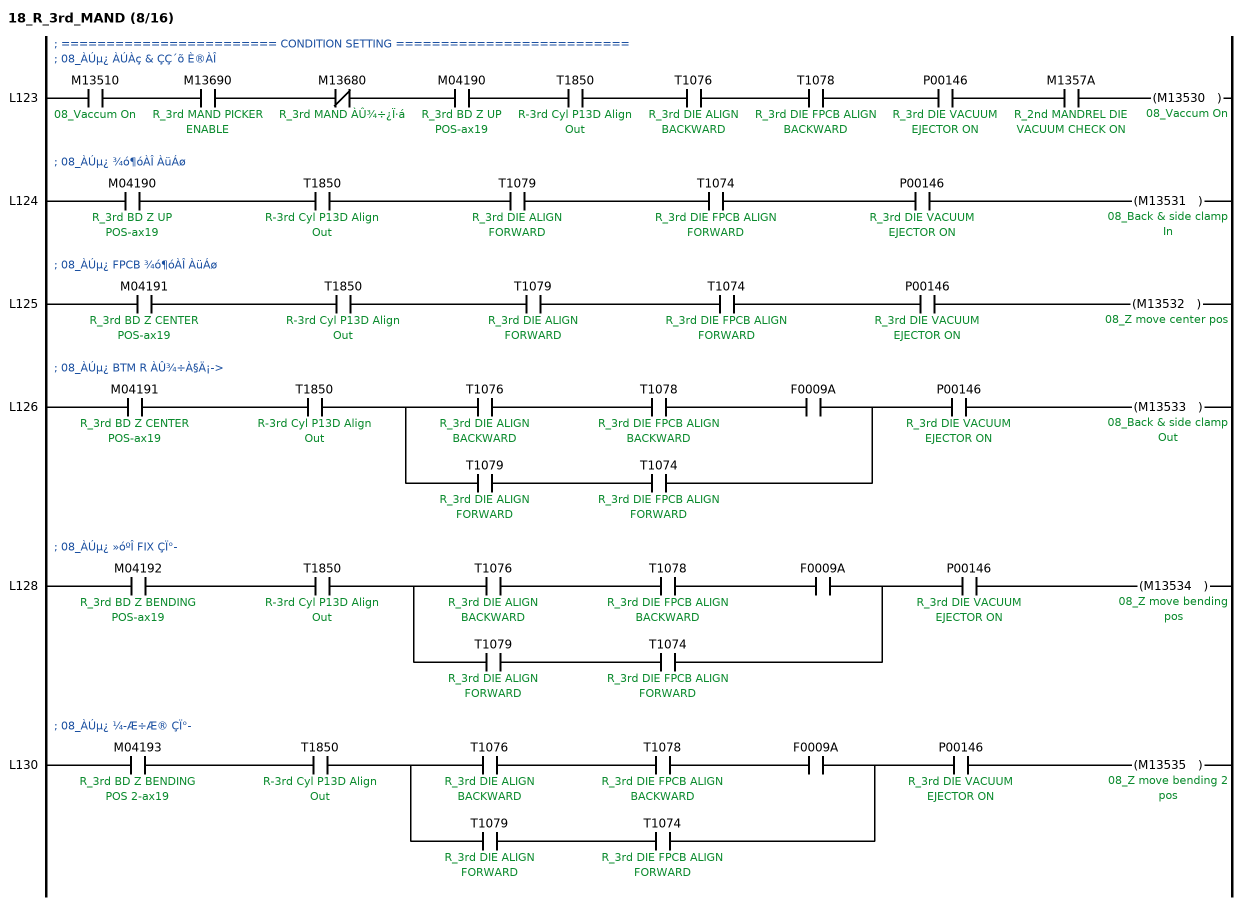
[picture p168: 18_R_3rd_MAND rungs L123-L130]
// ======================== CONDITION SETTING ==========================
; L123
LOAD      M13510	// 08_Vaccum On
AND       M13690	// R_3rd MAND PICKER ENABLE
AND NOT   M13680	// R_3rd MAND ÀÛ¾÷¿Ï·á
AND       M04190	// R_3rd BD Z UP POS-ax19
AND       T1850	// R-3rd Cyl P13D Align Out
AND       T1076	// R_3rd DIE ALIGN BACKWARD
AND       T1078	// R_3rd DIE FPCB ALIGN BACKWARD
AND       P00146	// R_3rd DIE VACUUM EJECTOR ON
AND       M1357A	// R_2nd MANDREL DIE VACUUM CHECK ON
OUT       M13530	// 08_Vaccum On
// output comment: 08_ÀÚµ¿ ÀÚÀç & ÇÇ´õ È®ÀÎ
; L124
LOAD      M04190	// R_3rd BD Z UP POS-ax19
AND       T1850	// R-3rd Cyl P13D Align Out
AND       T1079	// R_3rd DIE ALIGN FORWARD
AND       T1074	// R_3rd DIE FPCB ALIGN FORWARD
AND       P00146	// R_3rd DIE VACUUM EJECTOR ON
OUT       M13531	// 08_Back & side clamp In
// output comment: 08_ÀÚµ¿ ¾ó¶óÀÎ ÀüÁø
; L125
LOAD      M04191	// R_3rd BD Z CENTER POS-ax19
AND       T1850	// R-3rd Cyl P13D Align Out
AND       T1079	// R_3rd DIE ALIGN FORWARD
AND       T1074	// R_3rd DIE FPCB ALIGN FORWARD
AND       P00146	// R_3rd DIE VACUUM EJECTOR ON
OUT       M13532	// 08_Z move center pos
// output comment: 08_ÀÚµ¿ FPCB ¾ó¶óÀÎ ÀüÁø
; L126
LOAD      M04191	// R_3rd BD Z CENTER POS-ax19
AND       T1850	// R-3rd Cyl P13D Align Out
LOAD      T1076	// R_3rd DIE ALIGN BACKWARD
AND       T1078	// R_3rd DIE FPCB ALIGN BACKWARD
AND       F0009A
LOAD      T1079	// R_3rd DIE ALIGN FORWARD
AND       T1074	// R_3rd DIE FPCB ALIGN FORWARD
OR LOAD
AND LOAD
AND       P00146	// R_3rd DIE VACUUM EJECTOR ON
OUT       M13533	// 08_Back & side clamp Out
// output comment: 08_ÀÚµ¿ BTM R ÀÛ¾÷À§Ä¡->
; L128
LOAD      M04192	// R_3rd BD Z BENDING POS-ax19
AND       T1850	// R-3rd Cyl P13D Align Out
LOAD      T1076	// R_3rd DIE ALIGN BACKWARD
AND       T1078	// R_3rd DIE FPCB ALIGN BACKWARD
AND       F0009A
LOAD      T1079	// R_3rd DIE ALIGN FORWARD
AND       T1074	// R_3rd DIE FPCB ALIGN FORWARD
OR LOAD
AND LOAD
AND       P00146	// R_3rd DIE VACUUM EJECTOR ON
OUT       M13534	// 08_Z move bending pos
// output comment: 08_ÀÚµ¿ »óºÎ FIX ÇÏ°­
; L130
LOAD      M04193	// R_3rd BD Z BENDING POS 2-ax19
AND       T1850	// R-3rd Cyl P13D Align Out
LOAD      T1076	// R_3rd DIE ALIGN BACKWARD
AND       T1078	// R_3rd DIE FPCB ALIGN BACKWARD
AND       F0009A
LOAD      T1079	// R_3rd DIE ALIGN FORWARD
AND       T1074	// R_3rd DIE FPCB ALIGN FORWARD
OR LOAD
AND LOAD
AND       P00146	// R_3rd DIE VACUUM EJECTOR ON
OUT       M13535	// 08_Z move bending 2 pos
// output comment: 08_ÀÚµ¿ ¼­Æ÷Æ® ÇÏ°­

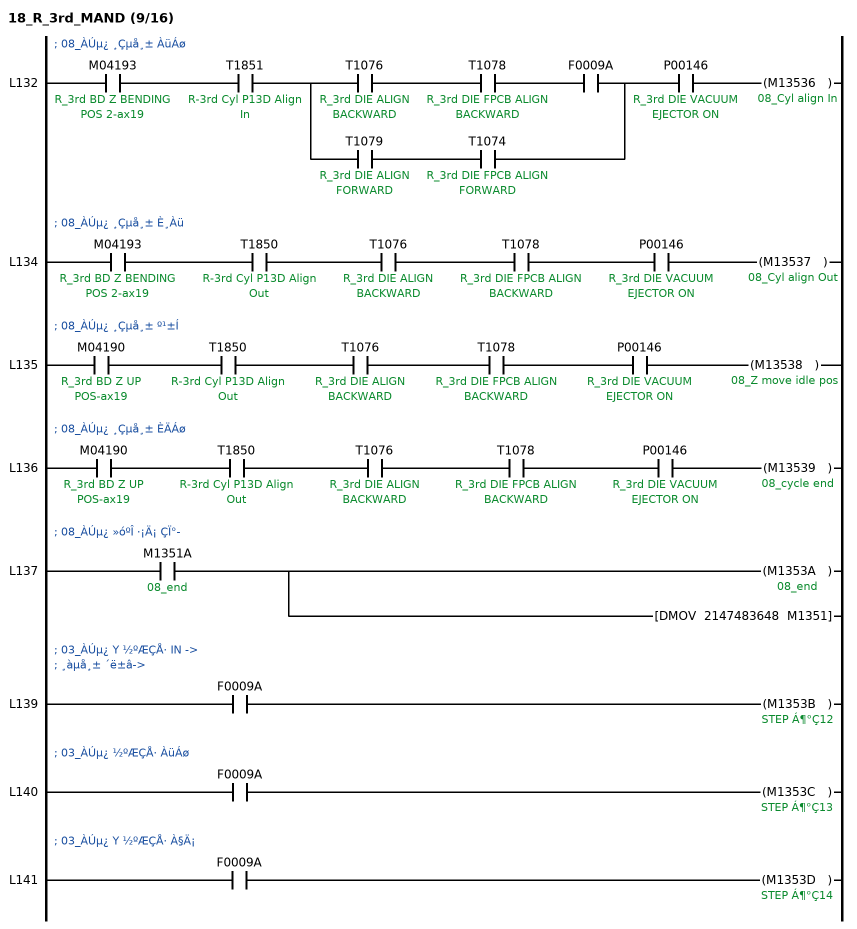
; L132
LOAD      M04193	// R_3rd BD Z BENDING POS 2-ax19
AND       T1851	// R-3rd Cyl P13D Align In
LOAD      T1076	// R_3rd DIE ALIGN BACKWARD
AND       T1078	// R_3rd DIE FPCB ALIGN BACKWARD
AND       F0009A
LOAD      T1079	// R_3rd DIE ALIGN FORWARD
AND       T1074	// R_3rd DIE FPCB ALIGN FORWARD
OR LOAD
AND LOAD
AND       P00146	// R_3rd DIE VACUUM EJECTOR ON
OUT       M13536	// 08_Cyl align In
// output comment: 08_ÀÚµ¿ ¸Çµå¸± ÀüÁø
; L134
LOAD      M04193	// R_3rd BD Z BENDING POS 2-ax19
AND       T1850	// R-3rd Cyl P13D Align Out
AND       T1076	// R_3rd DIE ALIGN BACKWARD
AND       T1078	// R_3rd DIE FPCB ALIGN BACKWARD
AND       P00146	// R_3rd DIE VACUUM EJECTOR ON
OUT       M13537	// 08_Cyl align Out
// output comment: 08_ÀÚµ¿ ¸Çµå¸± È¸Àü
; L135
LOAD      M04190	// R_3rd BD Z UP POS-ax19
AND       T1850	// R-3rd Cyl P13D Align Out
AND       T1076	// R_3rd DIE ALIGN BACKWARD
AND       T1078	// R_3rd DIE FPCB ALIGN BACKWARD
AND       P00146	// R_3rd DIE VACUUM EJECTOR ON
OUT       M13538	// 08_Z move idle pos
// output comment: 08_ÀÚµ¿ ¸Çµå¸± º¹±Í
; L136
LOAD      M04190	// R_3rd BD Z UP POS-ax19
AND       T1850	// R-3rd Cyl P13D Align Out
AND       T1076	// R_3rd DIE ALIGN BACKWARD
AND       T1078	// R_3rd DIE FPCB ALIGN BACKWARD
AND       P00146	// R_3rd DIE VACUUM EJECTOR ON
OUT       M13539	// 08_cycle end
// output comment: 08_ÀÚµ¿ ¸Çµå¸± ÈÄÁø
; L137
LOAD      M1351A	// 08_end
OUT       M1353A	// 08_end
DMOV      2147483648 M1351
// output comment: 08_ÀÚµ¿ »óºÎ ·¡Ä¡ ÇÏ°­
; L139
LOAD      F0009A
OUT       M1353B	// STEP Á¶°Ç12
// output comment: 03_ÀÚµ¿ Y ½ºÆÇÅ· IN -> ¸àµå¸± ´ë±â->
; L140
LOAD      F0009A
OUT       M1353C	// STEP Á¶°Ç13
// output comment: 03_ÀÚµ¿ ½ºÆÇÅ· ÀüÁø
; L141
LOAD      F0009A
OUT       M1353D	// STEP Á¶°Ç14
// output comment: 03_ÀÚµ¿ Y ½ºÆÇÅ· À§Ä¡

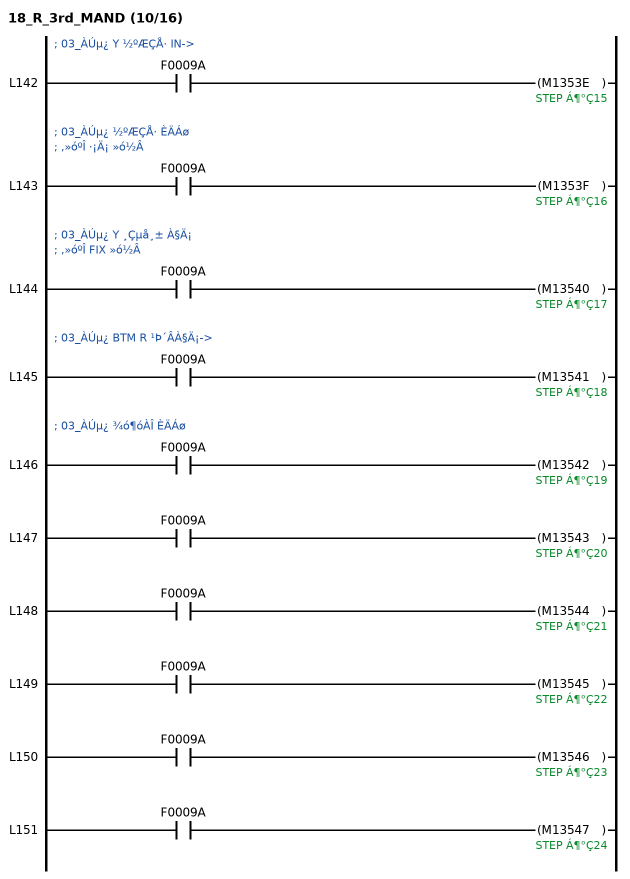
; L142
LOAD      F0009A
OUT       M1353E	// STEP Á¶°Ç15
// output comment: 03_ÀÚµ¿ Y ½ºÆÇÅ· IN->
; L143
LOAD      F0009A
OUT       M1353F	// STEP Á¶°Ç16
// output comment: 03_ÀÚµ¿ ½ºÆÇÅ· ÈÄÁø ,»óºÎ ·¡Ä¡ »ó½Â
; L144
LOAD      F0009A
OUT       M13540	// STEP Á¶°Ç17
// output comment: 03_ÀÚµ¿ Y ¸Çµå¸± À§Ä¡ ,»óºÎ FIX »ó½Â
; L145
LOAD      F0009A
OUT       M13541	// STEP Á¶°Ç18
// output comment: 03_ÀÚµ¿ BTM R ¹Þ´ÂÀ§Ä¡->
; L146
LOAD      F0009A
OUT       M13542	// STEP Á¶°Ç19
// output comment: 03_ÀÚµ¿ ¾ó¶óÀÎ ÈÄÁø
; L147
LOAD      F0009A
OUT       M13543	// STEP Á¶°Ç20
; L148
LOAD      F0009A
OUT       M13544	// STEP Á¶°Ç21
; L149
LOAD      F0009A
OUT       M13545	// STEP Á¶°Ç22
; L150
LOAD      F0009A
OUT       M13546	// STEP Á¶°Ç23
; L151
LOAD      F0009A
OUT       M13547	// STEP Á¶°Ç24

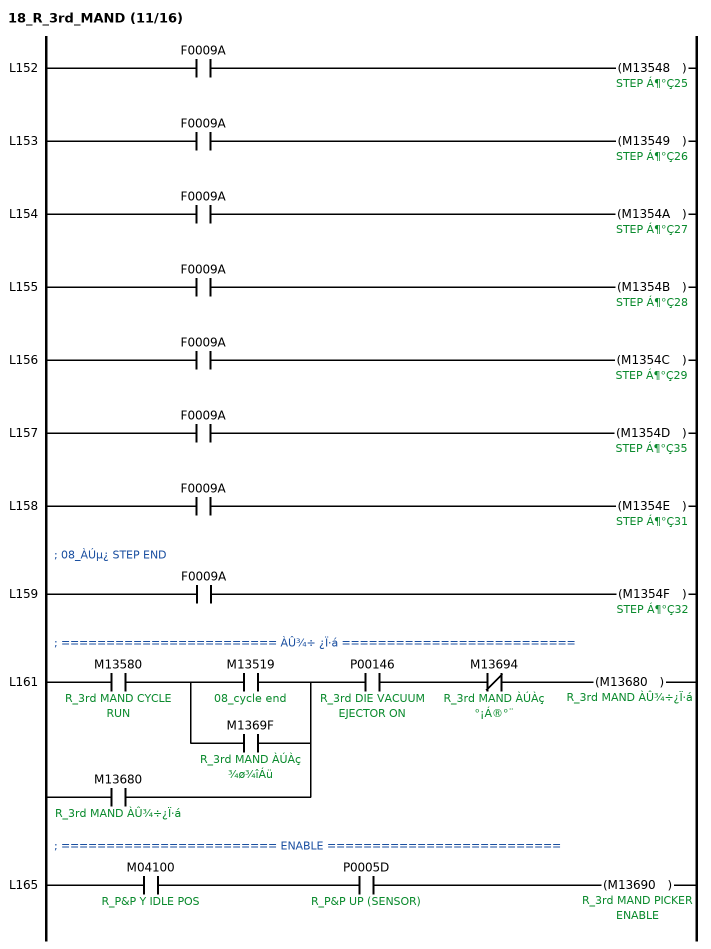
; L152
LOAD      F0009A
OUT       M13548	// STEP Á¶°Ç25
; L153
LOAD      F0009A
OUT       M13549	// STEP Á¶°Ç26
; L154
LOAD      F0009A
OUT       M1354A	// STEP Á¶°Ç27
; L155
LOAD      F0009A
OUT       M1354B	// STEP Á¶°Ç28
; L156
LOAD      F0009A
OUT       M1354C	// STEP Á¶°Ç29
; L157
LOAD      F0009A
OUT       M1354D	// STEP Á¶°Ç35
; L158
LOAD      F0009A
OUT       M1354E	// STEP Á¶°Ç31
; L159
LOAD      F0009A
OUT       M1354F	// STEP Á¶°Ç32
// output comment: 08_ÀÚµ¿ STEP END
// ======================== ÀÛ¾÷ ¿Ï·á ==========================
; L161
LOAD      M13580	// R_3rd MAND CYCLE RUN
LOAD      M13519	// 08_cycle end
OR        M1369F	// R_3rd MAND ÀÚÀç ¾ø¾îÁü
AND LOAD
OR        M13680	// R_3rd MAND ÀÛ¾÷¿Ï·á
AND       P00146	// R_3rd DIE VACUUM EJECTOR ON
AND NOT   M13694	// R_3rd MAND ÀÚÀç °¡Á®°¨
OUT       M13680	// R_3rd MAND ÀÛ¾÷¿Ï·á
// ======================== ENABLE ==========================
; L165
LOAD      M04100	// R_P&P Y IDLE POS
AND       P0005D	// R_P&P UP (SENSOR)
OUT       M13690	// R_3rd MAND PICKER ENABLE

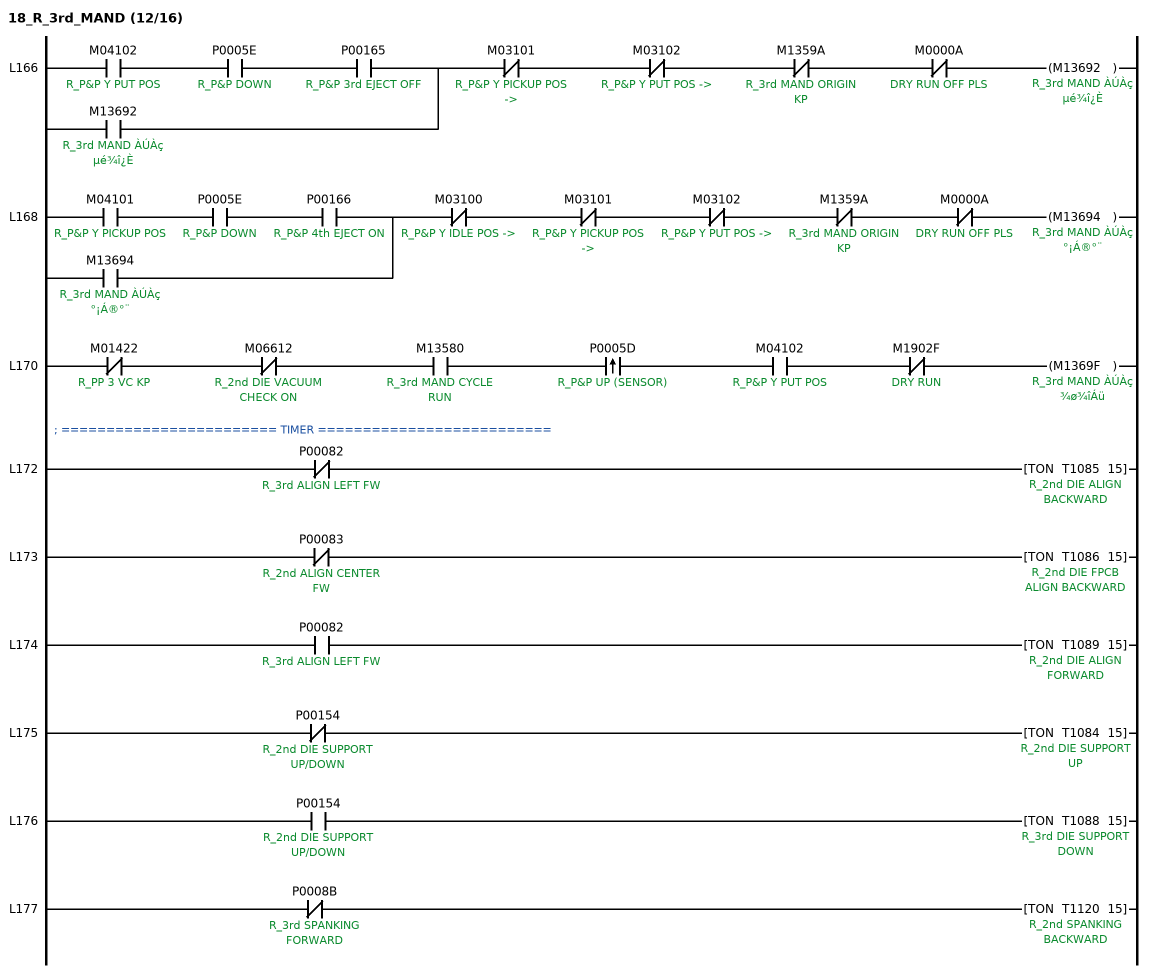
; L166
LOAD      M04102	// R_P&P Y PUT POS
AND       P0005E	// R_P&P DOWN
AND       P00165	// R_P&P 3rd EJECT OFF
OR        M13692	// R_3rd MAND ÀÚÀç µé¾î¿È
AND NOT   M03101	// R_P&P Y PICKUP POS ->
AND NOT   M03102	// R_P&P Y PUT POS ->
AND NOT   M1359A	// R_3rd MAND ORIGIN KP
AND NOT   M0000A	// DRY RUN OFF PLS
OUT       M13692	// R_3rd MAND ÀÚÀç µé¾î¿È
; L168
LOAD      M04101	// R_P&P Y PICKUP POS
AND       P0005E	// R_P&P DOWN
AND       P00166	// R_P&P 4th EJECT ON
OR        M13694	// R_3rd MAND ÀÚÀç °¡Á®°¨
AND NOT   M03100	// R_P&P Y IDLE POS ->
AND NOT   M03101	// R_P&P Y PICKUP POS ->
AND NOT   M03102	// R_P&P Y PUT POS ->
AND NOT   M1359A	// R_3rd MAND ORIGIN KP
AND NOT   M0000A	// DRY RUN OFF PLS
OUT       M13694	// R_3rd MAND ÀÚÀç °¡Á®°¨
; L170
LOAD NOT  M01422	// R_PP 3 VC KP
AND NOT   M06612	// R_2nd DIE VACUUM CHECK ON
AND       M13580	// R_3rd MAND CYCLE RUN
ANDP      P0005D	// R_P&P UP (SENSOR)
AND       M04102	// R_P&P Y PUT POS
AND NOT   M1902F	// DRY RUN
OUT       M1369F	// R_3rd MAND ÀÚÀç ¾ø¾îÁü
// ======================== TIMER ==========================
; L172
LOAD NOT  P00082	// R_3rd ALIGN LEFT FW
TON       T1085 15	// R_2nd DIE ALIGN BACKWARD
; L173
LOAD NOT  P00083	// R_2nd ALIGN CENTER FW
TON       T1086 15	// R_2nd DIE FPCB ALIGN BACKWARD
; L174
LOAD      P00082	// R_3rd ALIGN LEFT FW
TON       T1089 15	// R_2nd DIE ALIGN FORWARD
; L175
LOAD NOT  P00154	// R_2nd DIE SUPPORT UP/DOWN
TON       T1084 15	// R_2nd DIE SUPPORT UP
; L176
LOAD      P00154	// R_2nd DIE SUPPORT UP/DOWN
TON       T1088 15	// R_3rd DIE SUPPORT DOWN
; L177
LOAD NOT  P0008B	// R_3rd SPANKING FORWARD
TON       T1120 15	// R_2nd SPANKING BACKWARD

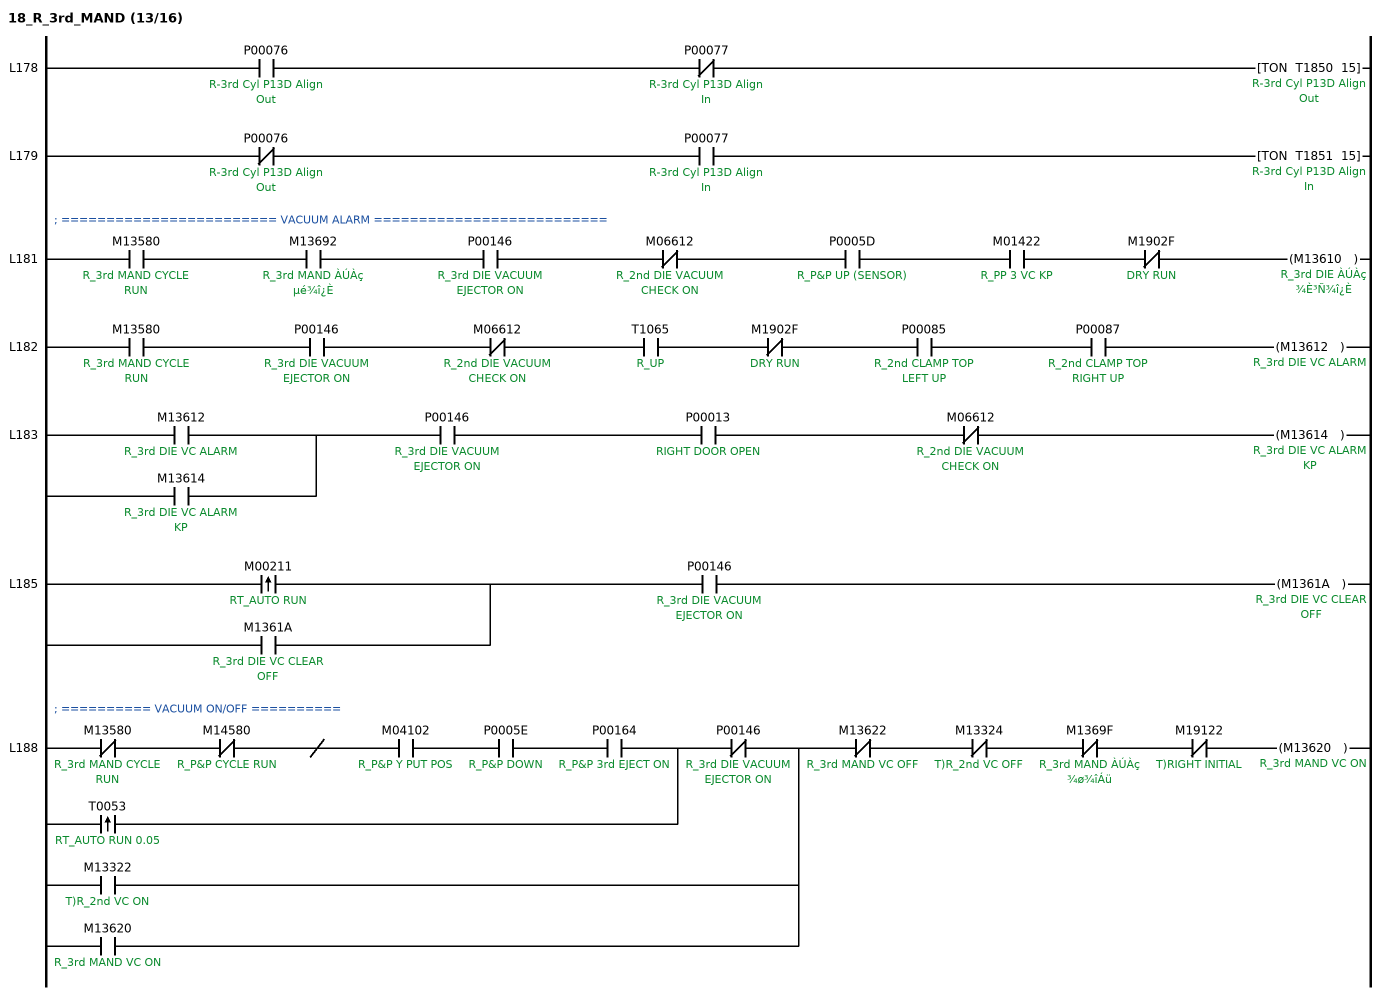
; L178
LOAD      P00076	// R-3rd Cyl P13D Align Out
AND NOT   P00077	// R-3rd Cyl P13D Align In
TON       T1850 15	// R-3rd Cyl P13D Align Out
; L179
LOAD NOT  P00076	// R-3rd Cyl P13D Align Out
AND       P00077	// R-3rd Cyl P13D Align In
TON       T1851 15	// R-3rd Cyl P13D Align In
// ======================== VACUUM ALARM ==========================
; L181
LOAD      M13580	// R_3rd MAND CYCLE RUN
AND       M13692	// R_3rd MAND ÀÚÀç µé¾î¿È
AND       P00146	// R_3rd DIE VACUUM EJECTOR ON
AND NOT   M06612	// R_2nd DIE VACUUM CHECK ON
AND       P0005D	// R_P&P UP (SENSOR)
AND       M01422	// R_PP 3 VC KP
AND NOT   M1902F	// DRY RUN
OUT       M13610	// R_3rd DIE ÀÚÀç ¾È³Ñ¾î¿È
; L182
LOAD      M13580	// R_3rd MAND CYCLE RUN
AND       P00146	// R_3rd DIE VACUUM EJECTOR ON
AND NOT   M06612	// R_2nd DIE VACUUM CHECK ON
AND       T1065	// R_UP
AND NOT   M1902F	// DRY RUN
AND       P00085	// R_2nd CLAMP TOP LEFT UP
AND       P00087	// R_2nd CLAMP TOP RIGHT UP
OUT       M13612	// R_3rd DIE VC ALARM
; L183
LOAD      M13612	// R_3rd DIE VC ALARM
OR        M13614	// R_3rd DIE VC ALARM KP
AND       P00146	// R_3rd DIE VACUUM EJECTOR ON
AND       P00013	// RIGHT DOOR OPEN
AND NOT   M06612	// R_2nd DIE VACUUM CHECK ON
OUT       M13614	// R_3rd DIE VC ALARM KP
; L185
LOADP     M00211	// RT_AUTO RUN
OR        M1361A	// R_3rd DIE VC CLEAR OFF
AND       P00146	// R_3rd DIE VACUUM EJECTOR ON
OUT       M1361A	// R_3rd DIE VC CLEAR OFF
// ========== VACUUM ON/OFF ==========
; L188
LOAD NOT  M13580	// R_3rd MAND CYCLE RUN
AND NOT   M14580	// R_P&P CYCLE RUN
NOT
AND       M04102	// R_P&P Y PUT POS
AND       P0005E	// R_P&P DOWN
AND       P00164	// R_P&P 3rd EJECT ON
ORP       T0053	// RT_AUTO RUN 0.05
AND NOT   P00146	// R_3rd DIE VACUUM EJECTOR ON
OR        M13322	// T)R_2nd VC ON
OR        M13620	// R_3rd MAND VC ON
AND NOT   M13622	// R_3rd MAND VC OFF
AND NOT   M13324	// T)R_2nd VC OFF
AND NOT   M1369F	// R_3rd MAND ÀÚÀç ¾ø¾îÁü
AND NOT   M19122	// T)RIGHT INITIAL
OUT       M13620	// R_3rd MAND VC ON

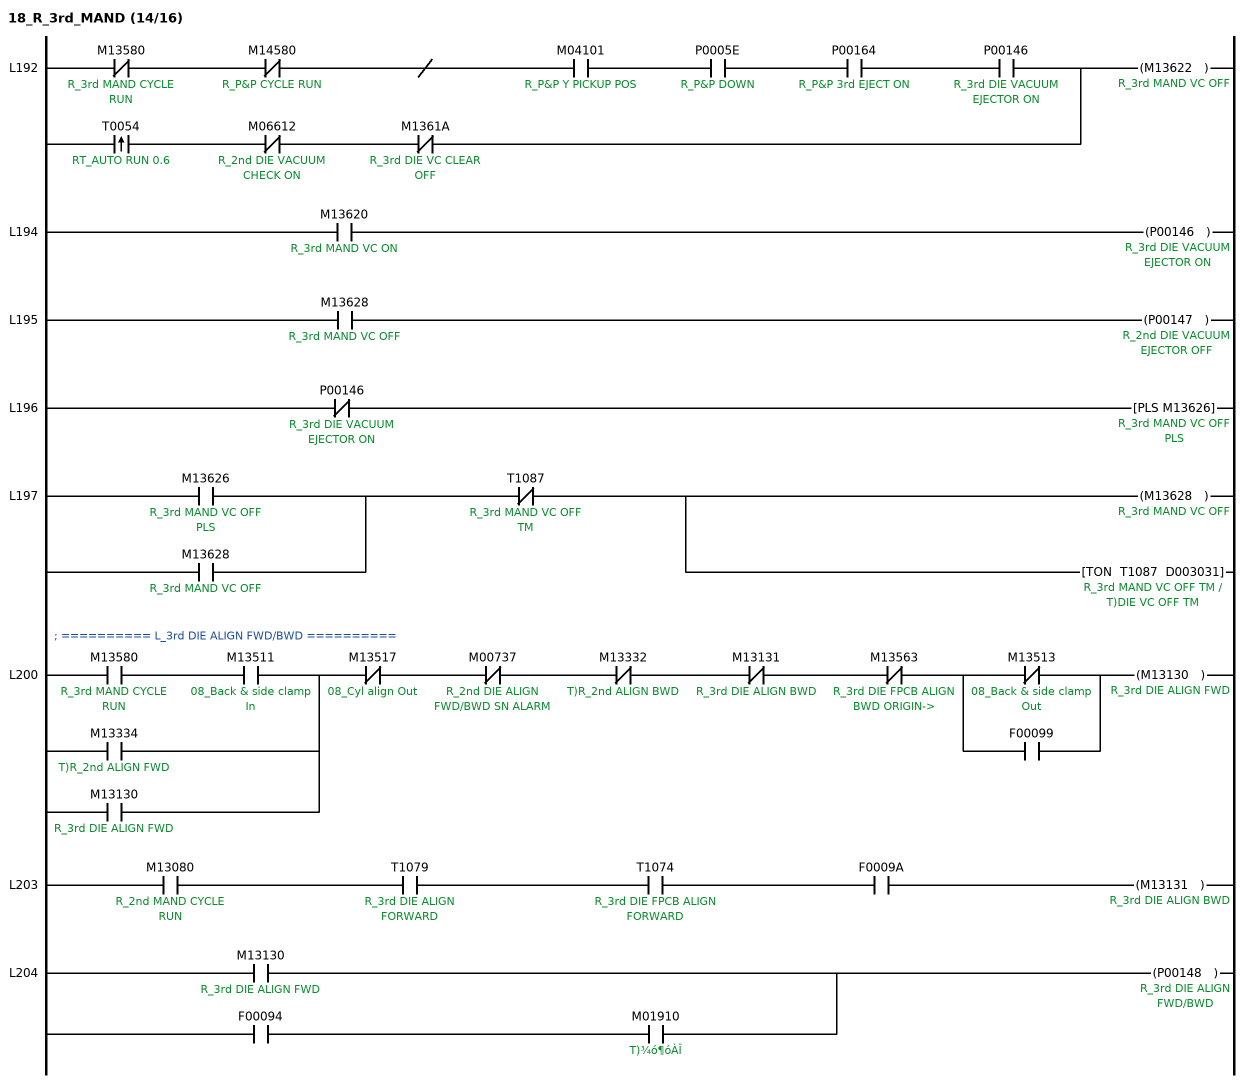
; L192
LOAD NOT  M13580	// R_3rd MAND CYCLE RUN
AND NOT   M14580	// R_P&P CYCLE RUN
NOT
AND       M04101	// R_P&P Y PICKUP POS
AND       P0005E	// R_P&P DOWN
AND       P00164	// R_P&P 3rd EJECT ON
AND       P00146	// R_3rd DIE VACUUM EJECTOR ON
LOADP     T0054	// RT_AUTO RUN 0.6
AND NOT   M06612	// R_2nd DIE VACUUM CHECK ON
AND NOT   M1361A	// R_3rd DIE VC CLEAR OFF
OR LOAD
OUT       M13622	// R_3rd MAND VC OFF
; L194
LOAD      M13620	// R_3rd MAND VC ON
OUT       P00146	// R_3rd DIE VACUUM EJECTOR ON
; L195
LOAD      M13628	// R_3rd MAND VC OFF
OUT       P00147	// R_2nd DIE VACUUM EJECTOR OFF
; L196
LOAD NOT  P00146	// R_3rd DIE VACUUM EJECTOR ON
OUTP      M13626	// R_3rd MAND VC OFF PLS
; L197
LOAD      M13626	// R_3rd MAND VC OFF PLS
OR        M13628	// R_3rd MAND VC OFF
AND NOT   T1087	// R_3rd MAND VC OFF TM
OUT       M13628	// R_3rd MAND VC OFF
TON       T1087 D003031	// R_3rd MAND VC OFF TM / T)DIE VC OFF TM
// ========== L_3rd DIE ALIGN FWD/BWD ==========
; L200
LOAD      M13580	// R_3rd MAND CYCLE RUN
AND       M13511	// 08_Back & side clamp In
OR        M13334	// T)R_2nd ALIGN FWD
OR        M13130	// R_3rd DIE ALIGN FWD
AND NOT   M13517	// 08_Cyl align Out
AND NOT   M00737	// R_2nd DIE ALIGN FWD/BWD SN ALARM
AND NOT   M13332	// T)R_2nd ALIGN BWD
AND NOT   M13131	// R_3rd DIE ALIGN BWD
AND NOT   M13563	// R_3rd DIE FPCB ALIGN BWD ORIGIN->
LOAD NOT  M13513	// 08_Back & side clamp Out
OR        F00099
AND LOAD
OUT       M13130	// R_3rd DIE ALIGN FWD
; L203
LOAD      M13080	// R_2nd MAND CYCLE RUN
AND       T1079	// R_3rd DIE ALIGN FORWARD
AND       T1074	// R_3rd DIE FPCB ALIGN FORWARD
AND       F0009A
OUT       M13131	// R_3rd DIE ALIGN BWD
; L204
LOAD      M13130	// R_3rd DIE ALIGN FWD
LOAD      F00094
AND       M01910	// T)¾ó¶óÀÎ
OR LOAD
OUT       P00148	// R_3rd DIE ALIGN FWD/BWD

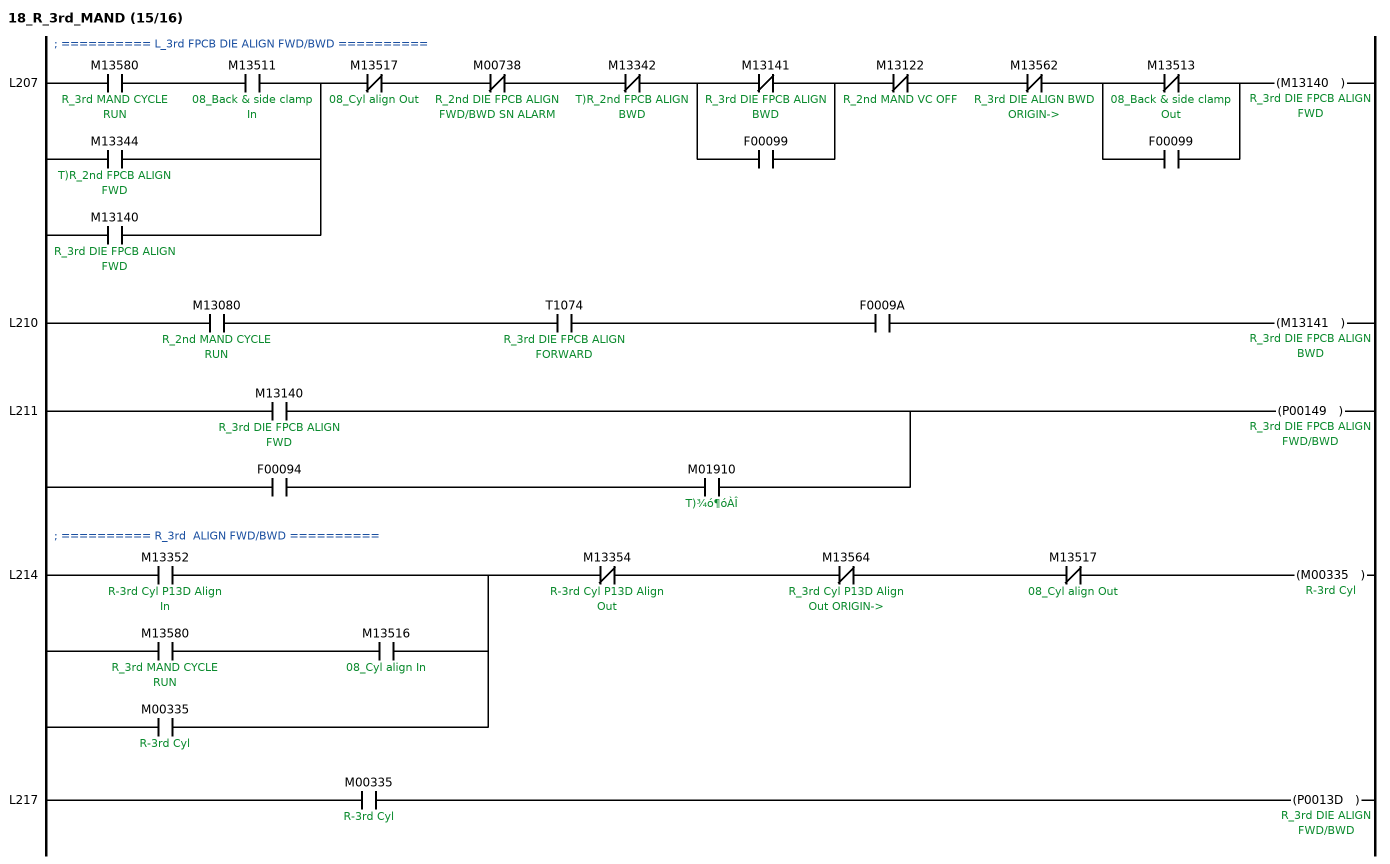
// ========== L_3rd FPCB DIE ALIGN FWD/BWD ==========
; L207
LOAD      M13580	// R_3rd MAND CYCLE RUN
AND       M13511	// 08_Back & side clamp In
OR        M13344	// T)R_2nd FPCB ALIGN FWD
OR        M13140	// R_3rd DIE FPCB ALIGN FWD
AND NOT   M13517	// 08_Cyl align Out
AND NOT   M00738	// R_2nd DIE FPCB ALIGN FWD/BWD SN ALARM
AND NOT   M13342	// T)R_2nd FPCB ALIGN BWD
LOAD NOT  M13141	// R_3rd DIE FPCB ALIGN BWD
OR        F00099
AND LOAD
AND NOT   M13122	// R_2nd MAND VC OFF
AND NOT   M13562	// R_3rd DIE ALIGN BWD ORIGIN->
LOAD NOT  M13513	// 08_Back & side clamp Out
OR        F00099
AND LOAD
OUT       M13140	// R_3rd DIE FPCB ALIGN FWD
; L210
LOAD      M13080	// R_2nd MAND CYCLE RUN
AND       T1074	// R_3rd DIE FPCB ALIGN FORWARD
AND       F0009A
OUT       M13141	// R_3rd DIE FPCB ALIGN BWD
; L211
LOAD      M13140	// R_3rd DIE FPCB ALIGN FWD
LOAD      F00094
AND       M01910	// T)¾ó¶óÀÎ
OR LOAD
OUT       P00149	// R_3rd DIE FPCB ALIGN FWD/BWD
// ========== R_3rd  ALIGN FWD/BWD ==========
; L214
LOAD      M13352	// R-3rd Cyl P13D Align In
LOAD      M13580	// R_3rd MAND CYCLE RUN
AND       M13516	// 08_Cyl align In
OR LOAD
OR        M00335	// R-3rd Cyl
AND NOT   M13354	// R-3rd Cyl P13D Align Out
AND NOT   M13564	// R_3rd Cyl P13D Align Out ORIGIN->
AND NOT   M13517	// 08_Cyl align Out
OUT       M00335	// R-3rd Cyl
; L217
LOAD      M00335	// R-3rd Cyl
OUT       P0013D	// R_3rd DIE ALIGN FWD/BWD

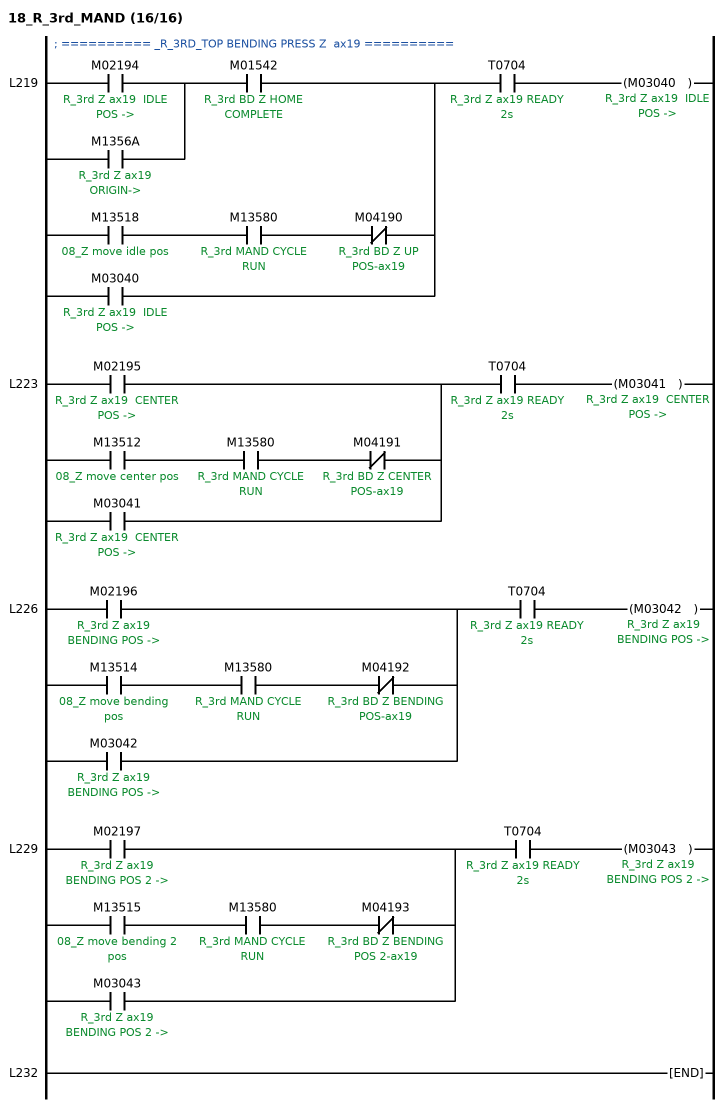
// ========== _R_3RD_TOP BENDING PRESS Z  ax19 ==========
; L219
LOAD      M02194	// R_3rd Z ax19  IDLE POS ->
OR        M1356A	// R_3rd Z ax19 ORIGIN->
AND       M01542	// R_3rd BD Z HOME COMPLETE
LOAD      M13518	// 08_Z move idle pos
AND       M13580	// R_3rd MAND CYCLE RUN
AND NOT   M04190	// R_3rd BD Z UP POS-ax19
OR LOAD
OR        M03040	// R_3rd Z ax19  IDLE POS ->
AND       T0704	// R_3rd Z ax19 READY 2s
OUT       M03040	// R_3rd Z ax19  IDLE POS ->
; L223
LOAD      M02195	// R_3rd Z ax19  CENTER POS ->
LOAD      M13512	// 08_Z move center pos
AND       M13580	// R_3rd MAND CYCLE RUN
AND NOT   M04191	// R_3rd BD Z CENTER POS-ax19
OR LOAD
OR        M03041	// R_3rd Z ax19  CENTER POS ->
AND       T0704	// R_3rd Z ax19 READY 2s
OUT       M03041	// R_3rd Z ax19  CENTER POS ->
; L226
LOAD      M02196	// R_3rd Z ax19 BENDING POS ->
LOAD      M13514	// 08_Z move bending pos
AND       M13580	// R_3rd MAND CYCLE RUN
AND NOT   M04192	// R_3rd BD Z BENDING POS-ax19
OR LOAD
OR        M03042	// R_3rd Z ax19  BENDING POS ->
AND       T0704	// R_3rd Z ax19 READY 2s
OUT       M03042	// R_3rd Z ax19  BENDING POS ->
; L229
LOAD      M02197	// R_3rd Z ax19 BENDING POS 2 ->
LOAD      M13515	// 08_Z move bending 2 pos
AND       M13580	// R_3rd MAND CYCLE RUN
AND NOT   M04193	// R_3rd BD Z BENDING POS 2-ax19
OR LOAD
OR        M03043	// R_3rd Z ax19 BENDING POS 2 ->
AND       T0704	// R_3rd Z ax19 READY 2s
OUT       M03043	// R_3rd Z ax19 BENDING POS 2 ->
; L232
END

PROGRAM 19_R_TOOL (task: ½ºÄµ ÇÁ·Î±×·¥)

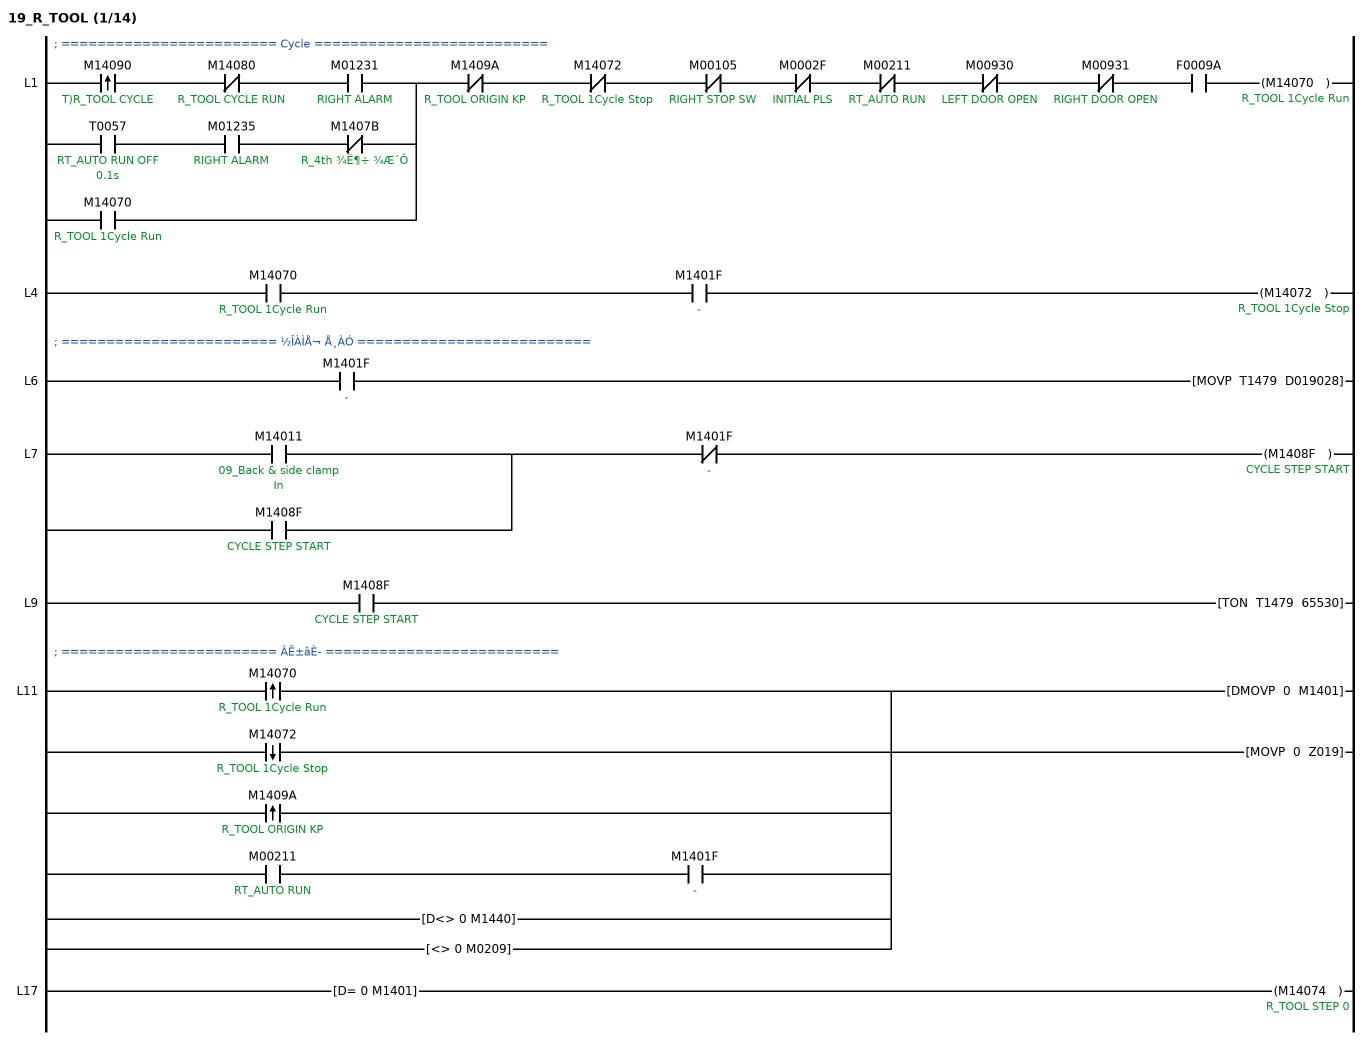
// ======================== Cycle ==========================
; L1
LOADP     M14090	// T)R_TOOL CYCLE
AND NOT   M14080	// R_TOOL CYCLE RUN
AND       M01231	// RIGHT ALARM
LOAD      T0057	// RT_AUTO RUN OFF 0.1s
AND       M01235	// RIGHT ALARM
AND NOT   M1407B	// R_4th ¾Ë¶÷ ¾Æ´Ô
OR LOAD
OR        M14070	// R_TOOL 1Cycle Run
AND NOT   M1409A	// R_TOOL ORIGIN KP
AND NOT   M14072	// R_TOOL 1Cycle Stop
AND NOT   M00105	// RIGHT STOP SW
AND NOT   M0002F	// INITIAL PLS
AND NOT   M00211	// RT_AUTO RUN
AND NOT   M00930	// LEFT DOOR OPEN
AND NOT   M00931	// RIGHT DOOR OPEN
AND       F0009A
OUT       M14070	// R_TOOL 1Cycle Run
; L4
LOAD      M14070	// R_TOOL 1Cycle Run
AND       M1401F	// -
OUT       M14072	// R_TOOL 1Cycle Stop
// ======================== ½ÎÀÌÅ¬ Å¸ÀÓ ==========================
; L6
LOAD      M1401F	// -
MOVP      T1479 D019028
; L7
LOAD      M14011	// 09_Back & side clamp In
OR        M1408F	// CYCLE STEP START
AND NOT   M1401F	// -
OUT       M1408F	// CYCLE STEP START
; L9
LOAD      M1408F	// CYCLE STEP START
TON       T1479 65530
// ======================== ÃÊ±âÈ­ ==========================
; L11
LOADP     M14070	// R_TOOL 1Cycle Run
ORN       M14072	// R_TOOL 1Cycle Stop
ORP       M1409A	// R_TOOL ORIGIN KP
LOAD      M00211	// RT_AUTO RUN
AND       M1401F	// -
OR LOAD
ORD<>     0 M1440
OR<>      0 M0209
DMOVP     0 M1401
MOVP      0 Z019
; L17
LOADD=    0 M1401
OUT       M14074	// R_TOOL STEP 0

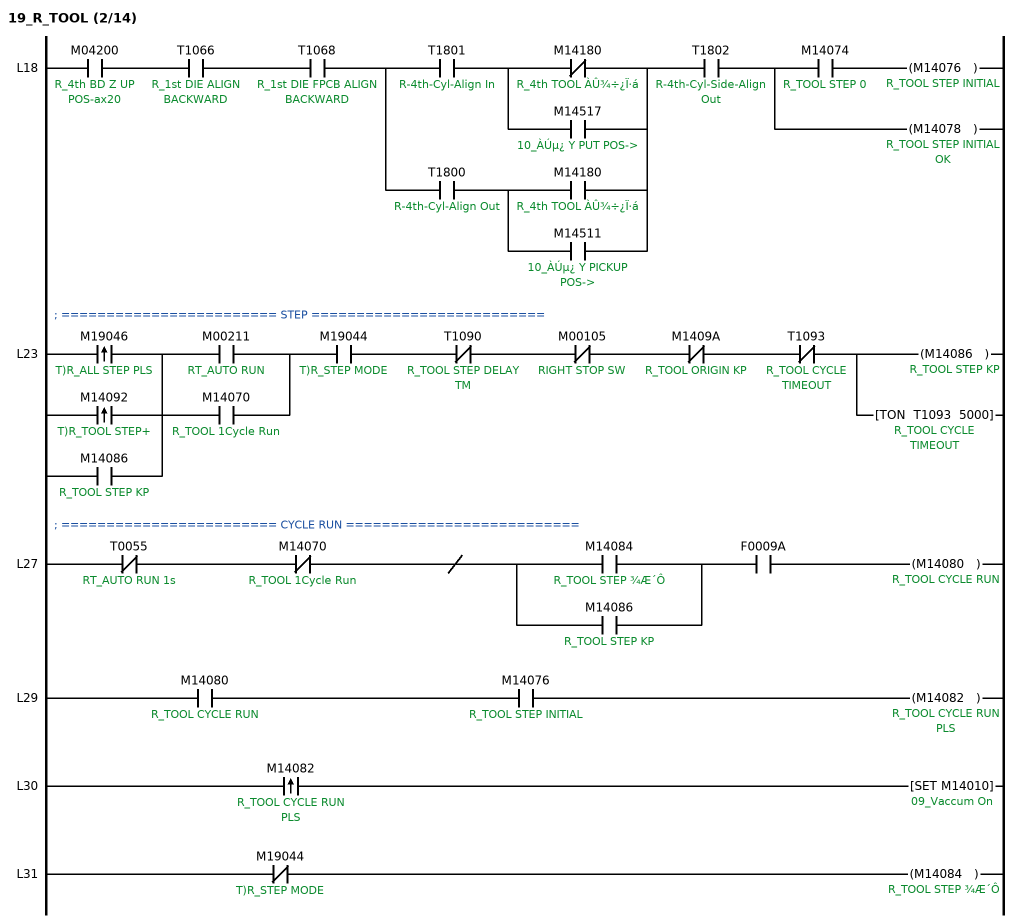
; L18
LOAD      M04200	// R_4th BD Z UP POS-ax20
AND       T1066	// R_1st DIE ALIGN BACKWARD
AND       T1068	// R_1st DIE FPCB ALIGN BACKWARD
LOAD      T1801	// R-4th-Cyl-Align In
LOAD NOT  M14180	// R_4th TOOL ÀÛ¾÷¿Ï·á
OR        M14517	// 10_ÀÚµ¿ Y PUT POS->
AND LOAD
LOAD      T1800	// R-4th-Cyl-Align Out
LOAD      M14180	// R_4th TOOL ÀÛ¾÷¿Ï·á
OR        M14511	// 10_ÀÚµ¿ Y PICKUP POS->
AND LOAD
OR LOAD
AND LOAD
AND       T1802	// R-4th-Cyl-Side-Align Out
MPUSH
AND       M14074	// R_TOOL STEP 0
OUT       M14076	// R_TOOL STEP INITIAL
MPOP
OUT       M14078	// R_TOOL STEP INITIAL OK
// ======================== STEP ==========================
; L23
LOADP     M19046	// T)R_ALL STEP PLS
ORP       M14092	// T)R_TOOL STEP+
OR        M14086	// R_TOOL STEP KP
LOAD      M00211	// RT_AUTO RUN
OR        M14070	// R_TOOL 1Cycle Run
AND LOAD
AND       M19044	// T)R_STEP MODE
AND NOT   T1090	// R_TOOL STEP DELAY TM
AND NOT   M00105	// RIGHT STOP SW
AND NOT   M1409A	// R_TOOL ORIGIN KP
AND NOT   T1093	// R_TOOL CYCLE TIMEOUT
OUT       M14086	// R_TOOL STEP KP
TON       T1093 5000	// R_TOOL CYCLE TIMEOUT
// ======================== CYCLE RUN ==========================
; L27
LOAD NOT  T0055	// RT_AUTO RUN 1s
AND NOT   M14070	// R_TOOL 1Cycle Run
NOT
LOAD      M14084	// R_TOOL STEP ¾Æ´Ô
OR        M14086	// R_TOOL STEP KP
AND LOAD
AND       F0009A
OUT       M14080	// R_TOOL CYCLE RUN
; L29
LOAD      M14080	// R_TOOL CYCLE RUN
AND       M14076	// R_TOOL STEP INITIAL
OUT       M14082	// R_TOOL CYCLE RUN PLS
; L30
LOADP     M14082	// R_TOOL CYCLE RUN PLS
SET       M14010	// 09_Vaccum On
; L31
LOAD NOT  M19044	// T)R_STEP MODE
OUT       M14084	// R_TOOL STEP ¾Æ´Ô

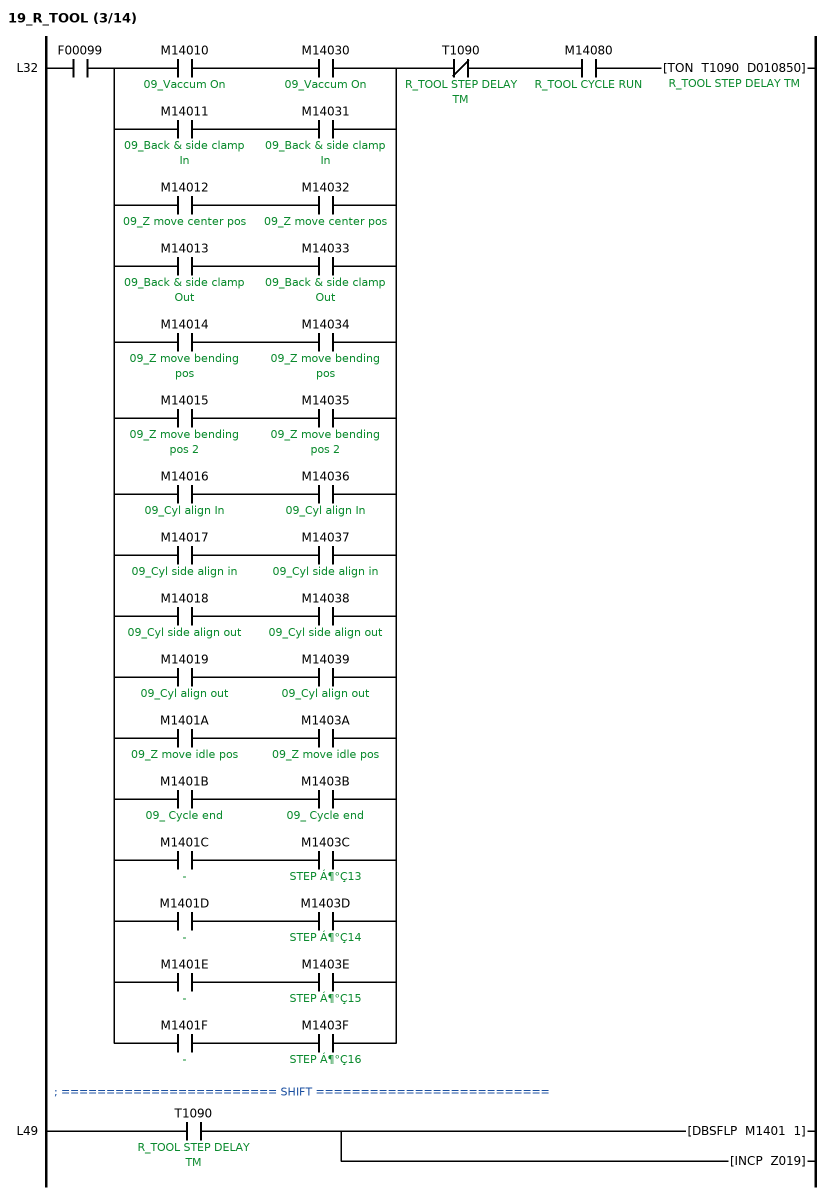
; L32
LOAD      F00099
LOAD      M14010	// 09_Vaccum On
AND       M14030	// 09_Vaccum On
LOAD      M14011	// 09_Back & side clamp In
AND       M14031	// 09_Back & side clamp In
OR LOAD
LOAD      M14012	// 09_Z move center pos
AND       M14032	// 09_Z move center pos
OR LOAD
LOAD      M14013	// 09_Back & side clamp Out
AND       M14033	// 09_Back & side clamp Out
OR LOAD
LOAD      M14014	// 09_Z move bending pos
AND       M14034	// 09_Z move bending pos
OR LOAD
LOAD      M14015	// 09_Z move bending pos 2
AND       M14035	// 09_Z move bending pos 2
OR LOAD
LOAD      M14016	// 09_Cyl align In
AND       M14036	// 09_Cyl align In
OR LOAD
LOAD      M14017	// 09_Cyl side align in
AND       M14037	// 09_Cyl side align in
OR LOAD
LOAD      M14018	// 09_Cyl side align out
AND       M14038	// 09_Cyl side align out
OR LOAD
LOAD      M14019	// 09_Cyl align out
AND       M14039	// 09_Cyl align out
OR LOAD
LOAD      M1401A	// 09_Z move idle pos
AND       M1403A	// 09_Z move idle pos
OR LOAD
LOAD      M1401B	// 09_ Cycle end
AND       M1403B	// 09_ Cycle end
OR LOAD
LOAD      M1401C	// -
AND       M1403C	// STEP Á¶°Ç13
OR LOAD
LOAD      M1401D	// -
AND       M1403D	// STEP Á¶°Ç14
OR LOAD
LOAD      M1401E	// -
AND       M1403E	// STEP Á¶°Ç15
OR LOAD
LOAD      M1401F	// -
AND       M1403F	// STEP Á¶°Ç16
OR LOAD
AND LOAD
AND NOT   T1090	// R_TOOL STEP DELAY TM
AND       M14080	// R_TOOL CYCLE RUN
TON       T1090 D010850	// R_TOOL STEP DELAY TM
// ======================== SHIFT ==========================
; L49
LOAD      T1090	// R_TOOL STEP DELAY TM
DBSFLP    M1401 1
INCP      Z019

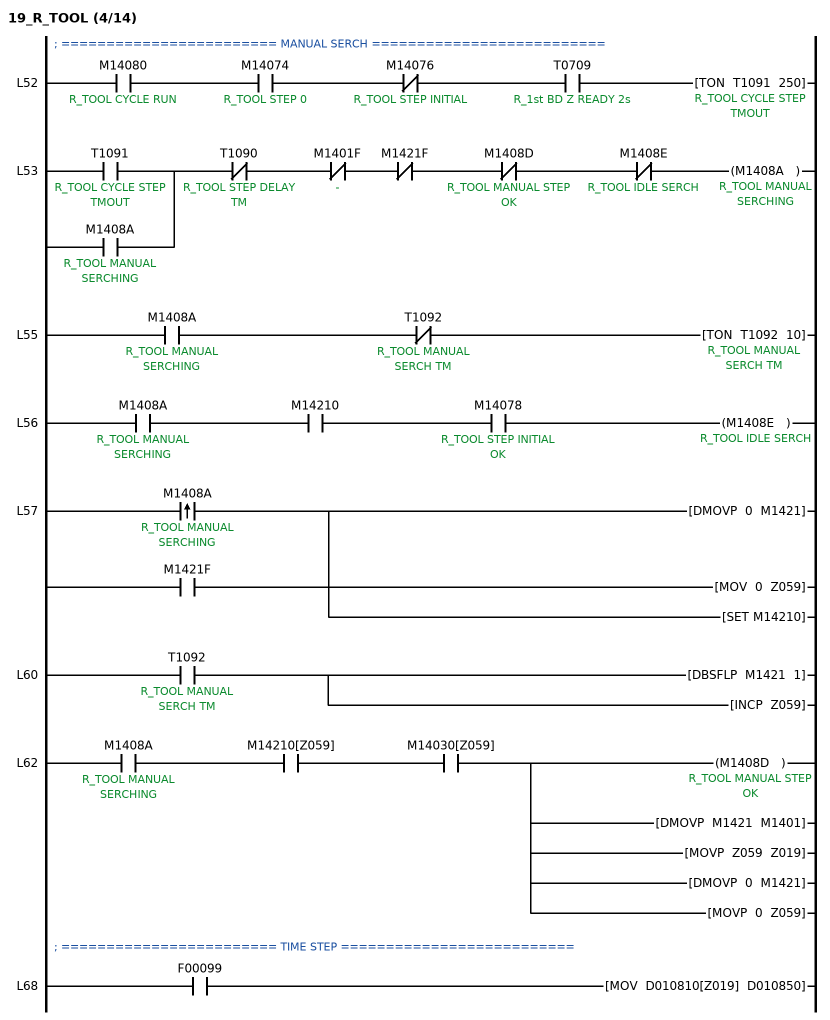
// ======================== MANUAL SERCH ==========================
; L52
LOAD      M14080	// R_TOOL CYCLE RUN
AND       M14074	// R_TOOL STEP 0
AND NOT   M14076	// R_TOOL STEP INITIAL
AND       T0709	// R_1st BD Z READY 2s
TON       T1091 250	// R_TOOL CYCLE STEP TMOUT
; L53
LOAD      T1091	// R_TOOL CYCLE STEP TMOUT
OR        M1408A	// R_TOOL MANUAL SERCHING
AND NOT   T1090	// R_TOOL STEP DELAY TM
AND NOT   M1401F	// -
AND NOT   M1421F
AND NOT   M1408D	// R_TOOL MANUAL STEP OK
AND NOT   M1408E	// R_TOOL IDLE SERCH
OUT       M1408A	// R_TOOL MANUAL SERCHING
; L55
LOAD      M1408A	// R_TOOL MANUAL SERCHING
AND NOT   T1092	// R_TOOL MANUAL SERCH TM
TON       T1092 10	// R_TOOL MANUAL SERCH TM
; L56
LOAD      M1408A	// R_TOOL MANUAL SERCHING
AND       M14210
AND       M14078	// R_TOOL STEP INITIAL OK
OUT       M1408E	// R_TOOL IDLE SERCH
; L57
LOADP     M1408A	// R_TOOL MANUAL SERCHING
OR        M1421F
DMOVP     0 M1421
MOV       0 Z059
SET       M14210
; L60
LOAD      T1092	// R_TOOL MANUAL SERCH TM
DBSFLP    M1421 1
INCP      Z059
; L62
LOAD      M1408A	// R_TOOL MANUAL SERCHING
AND       M14210[Z059]
AND       M14030[Z059]
OUT       M1408D	// R_TOOL MANUAL STEP OK
DMOVP     M1421 M1401
MOVP      Z059 Z019
DMOVP     0 M1421
MOVP      0 Z059
// ======================== TIME STEP ==========================
; L68
LOAD      F00099
MOV       D010810[Z019] D010850

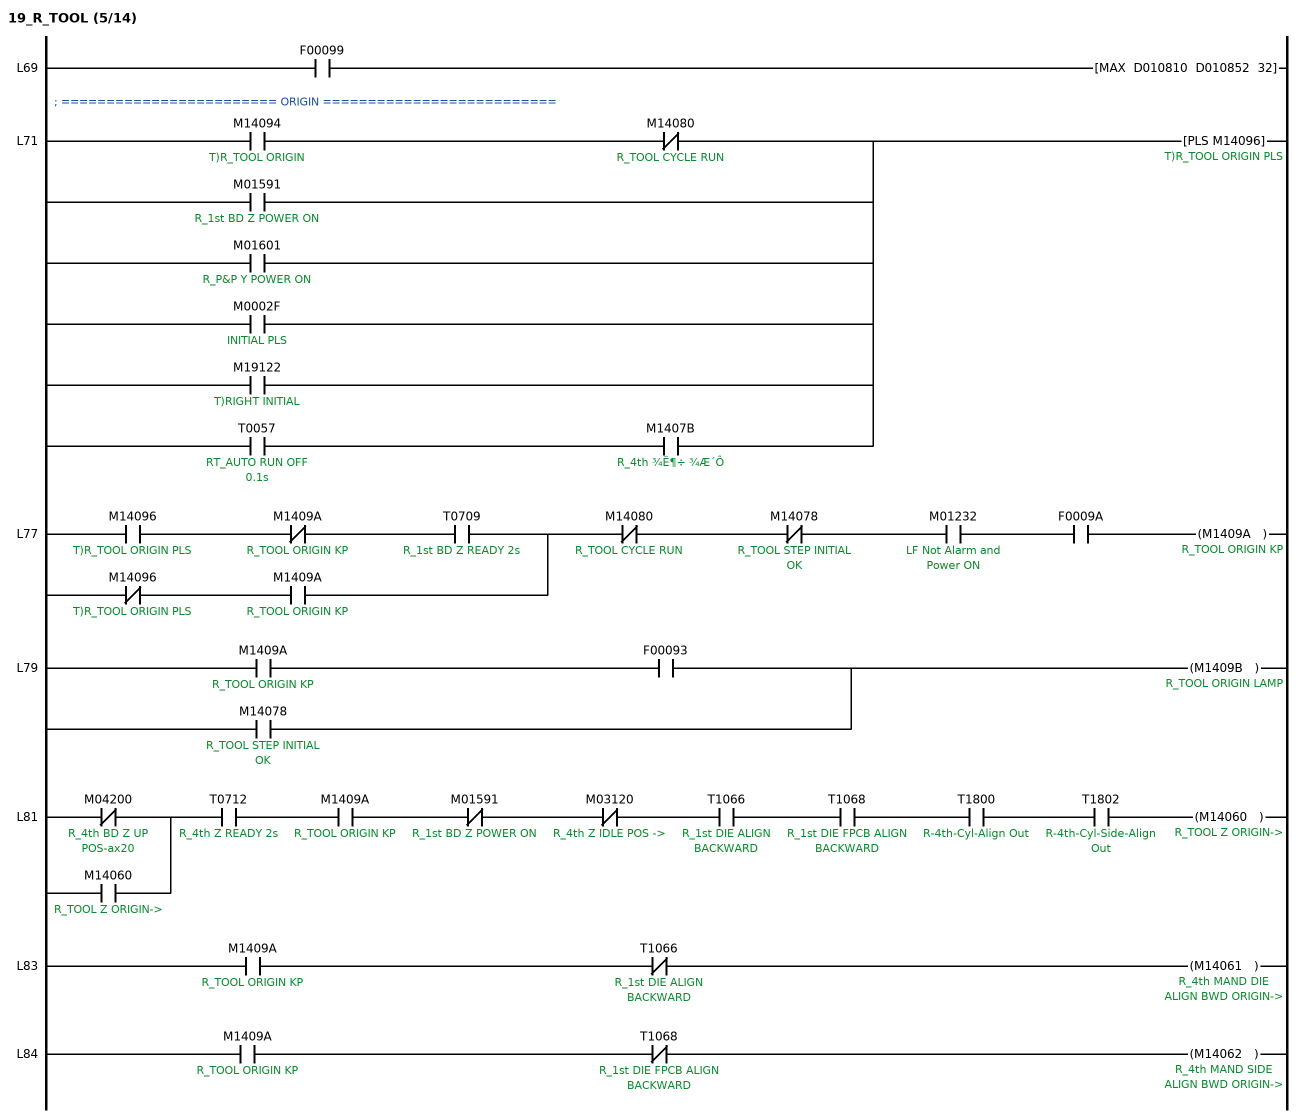
; L69
LOAD      F00099
MAX       D010810 D010852 32
// ======================== ORIGIN ==========================
; L71
LOAD      M14094	// T)R_TOOL ORIGIN
AND NOT   M14080	// R_TOOL CYCLE RUN
OR        M01591	// R_1st BD Z POWER ON
OR        M01601	// R_P&P Y POWER ON
OR        M0002F	// INITIAL PLS
OR        M19122	// T)RIGHT INITIAL
LOAD      T0057	// RT_AUTO RUN OFF 0.1s
AND       M1407B	// R_4th ¾Ë¶÷ ¾Æ´Ô
OR LOAD
OUTP      M14096	// T)R_TOOL ORIGIN PLS
; L77
LOAD      M14096	// T)R_TOOL ORIGIN PLS
AND NOT   M1409A	// R_TOOL ORIGIN KP
AND       T0709	// R_1st BD Z READY 2s
LOAD NOT  M14096	// T)R_TOOL ORIGIN PLS
AND       M1409A	// R_TOOL ORIGIN KP
OR LOAD
AND NOT   M14080	// R_TOOL CYCLE RUN
AND NOT   M14078	// R_TOOL STEP INITIAL OK
AND       M01232	// LF Not Alarm and Power ON
AND       F0009A
OUT       M1409A	// R_TOOL ORIGIN KP
; L79
LOAD      M1409A	// R_TOOL ORIGIN KP
AND       F00093
OR        M14078	// R_TOOL STEP INITIAL OK
OUT       M1409B	// R_TOOL ORIGIN LAMP
; L81
LOAD NOT  M04200	// R_4th BD Z UP POS-ax20
OR        M14060	// R_TOOL Z ORIGIN->
AND       T0712	// R_4th Z READY 2s
AND       M1409A	// R_TOOL ORIGIN KP
AND NOT   M01591	// R_1st BD Z POWER ON
AND NOT   M03120	// R_4th Z IDLE POS ->
AND       T1066	// R_1st DIE ALIGN BACKWARD
AND       T1068	// R_1st DIE FPCB ALIGN BACKWARD
AND       T1800	// R-4th-Cyl-Align Out
AND       T1802	// R-4th-Cyl-Side-Align Out
OUT       M14060	// R_TOOL Z ORIGIN->
; L83
LOAD      M1409A	// R_TOOL ORIGIN KP
AND NOT   T1066	// R_1st DIE ALIGN BACKWARD
OUT       M14061	// R_4th MAND DIE ALIGN BWD ORIGIN->
; L84
LOAD      M1409A	// R_TOOL ORIGIN KP
AND NOT   T1068	// R_1st DIE FPCB ALIGN BACKWARD
OUT       M14062	// R_4th MAND SIDE ALIGN BWD ORIGIN->

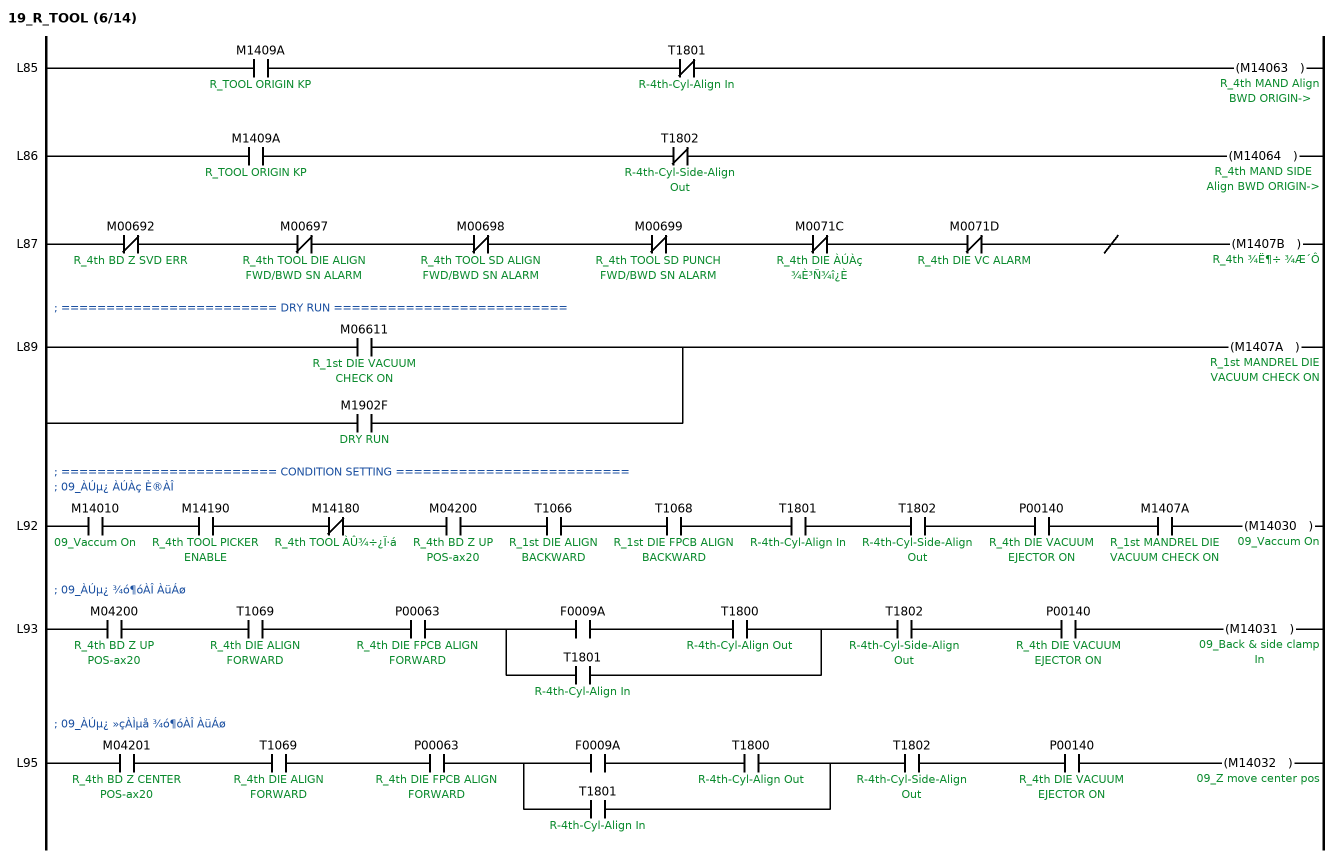
; L85
LOAD      M1409A	// R_TOOL ORIGIN KP
AND NOT   T1801	// R-4th-Cyl-Align In
OUT       M14063	// R_4th MAND Align BWD ORIGIN->
; L86
LOAD      M1409A	// R_TOOL ORIGIN KP
AND NOT   T1802	// R-4th-Cyl-Side-Align Out
OUT       M14064	// R_4th MAND SIDE Align BWD ORIGIN->
; L87
LOAD NOT  M00692	// R_4th BD Z SVD ERR
AND NOT   M00697	// R_4th TOOL DIE ALIGN FWD/BWD SN ALARM
AND NOT   M00698	// R_4th TOOL SD ALIGN FWD/BWD SN ALARM
AND NOT   M00699	// R_4th TOOL SD PUNCH FWD/BWD SN ALARM
AND NOT   M0071C	// R_4th DIE ÀÚÀç ¾È³Ñ¾î¿È
AND NOT   M0071D	// R_4th DIE VC ALARM
NOT
OUT       M1407B	// R_4th ¾Ë¶÷ ¾Æ´Ô
// ======================== DRY RUN ==========================
; L89
LOAD      M06611	// R_1st DIE VACUUM CHECK ON
OR        M1902F	// DRY RUN
OUT       M1407A	// R_1st MANDREL DIE VACUUM CHECK ON
// ======================== CONDITION SETTING ==========================
; L92
LOAD      M14010	// 09_Vaccum On
AND       M14190	// R_4th TOOL PICKER ENABLE
AND NOT   M14180	// R_4th TOOL ÀÛ¾÷¿Ï·á
AND       M04200	// R_4th BD Z UP POS-ax20
AND       T1066	// R_1st DIE ALIGN BACKWARD
AND       T1068	// R_1st DIE FPCB ALIGN BACKWARD
AND       T1801	// R-4th-Cyl-Align In
AND       T1802	// R-4th-Cyl-Side-Align Out
AND       P00140	// R_4th DIE VACUUM EJECTOR ON
AND       M1407A	// R_1st MANDREL DIE VACUUM CHECK ON
OUT       M14030	// 09_Vaccum On
// output comment: 09_ÀÚµ¿ ÀÚÀç È®ÀÎ
; L93
LOAD      M04200	// R_4th BD Z UP POS-ax20
AND       T1069	// R_4th DIE ALIGN FORWARD
AND       P00063	// R_4th DIE FPCB ALIGN FORWARD
LOAD      F0009A
AND       T1800	// R-4th-Cyl-Align Out
OR        T1801	// R-4th-Cyl-Align In
AND LOAD
AND       T1802	// R-4th-Cyl-Side-Align Out
AND       P00140	// R_4th DIE VACUUM EJECTOR ON
OUT       M14031	// 09_Back & side clamp In
// output comment: 09_ÀÚµ¿ ¾ó¶óÀÎ ÀüÁø
; L95
LOAD      M04201	// R_4th BD Z CENTER POS-ax20
AND       T1069	// R_4th DIE ALIGN FORWARD
AND       P00063	// R_4th DIE FPCB ALIGN FORWARD
LOAD      F0009A
AND       T1800	// R-4th-Cyl-Align Out
OR        T1801	// R-4th-Cyl-Align In
AND LOAD
AND       T1802	// R-4th-Cyl-Side-Align Out
AND       P00140	// R_4th DIE VACUUM EJECTOR ON
OUT       M14032	// 09_Z move center pos
// output comment: 09_ÀÚµ¿ »çÀÌµå ¾ó¶óÀÎ ÀüÁø

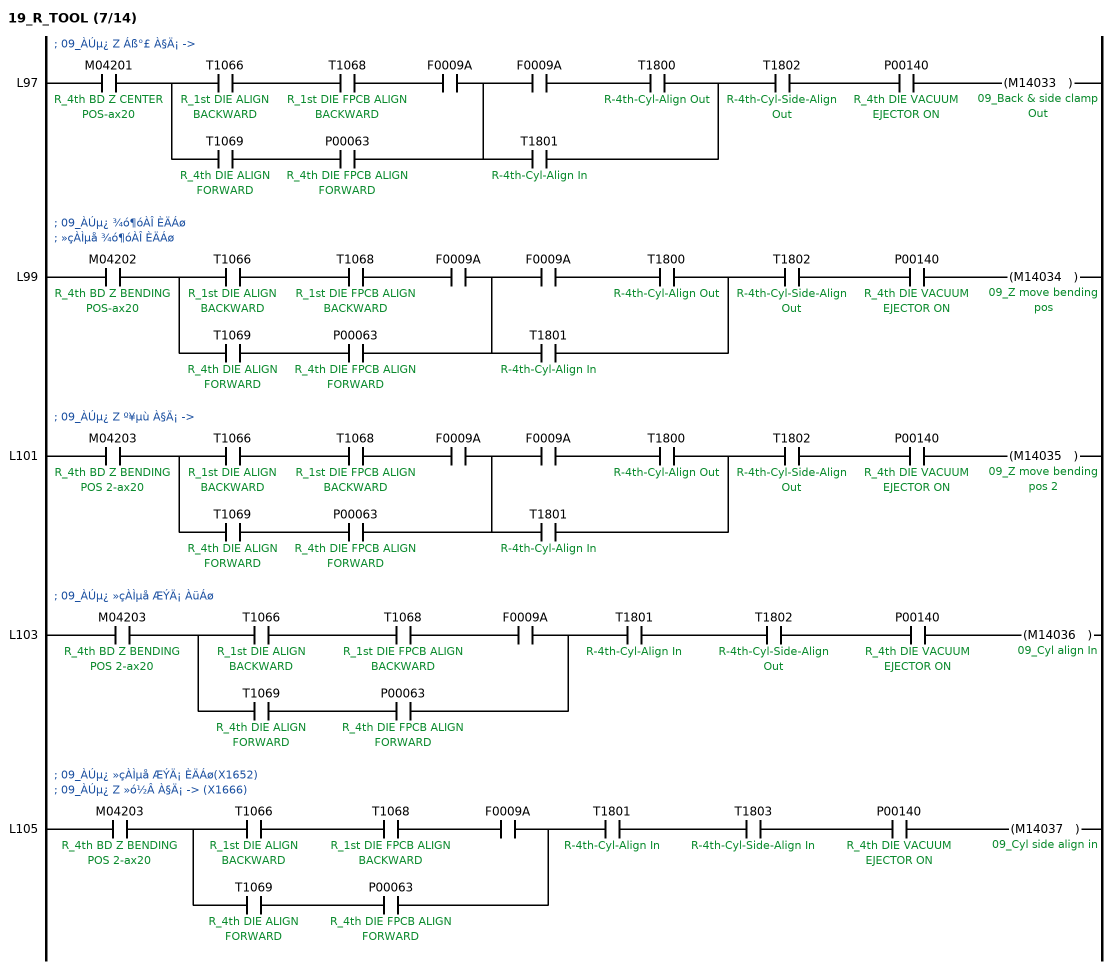
; L97
LOAD      M04201	// R_4th BD Z CENTER POS-ax20
LOAD      T1066	// R_1st DIE ALIGN BACKWARD
AND       T1068	// R_1st DIE FPCB ALIGN BACKWARD
AND       F0009A
LOAD      T1069	// R_4th DIE ALIGN FORWARD
AND       P00063	// R_4th DIE FPCB ALIGN FORWARD
OR LOAD
AND LOAD
LOAD      F0009A
AND       T1800	// R-4th-Cyl-Align Out
OR        T1801	// R-4th-Cyl-Align In
AND LOAD
AND       T1802	// R-4th-Cyl-Side-Align Out
AND       P00140	// R_4th DIE VACUUM EJECTOR ON
OUT       M14033	// 09_Back & side clamp Out
// output comment: 09_ÀÚµ¿ Z Áß°£ À§Ä¡ ->
; L99
LOAD      M04202	// R_4th BD Z BENDING POS-ax20
LOAD      T1066	// R_1st DIE ALIGN BACKWARD
AND       T1068	// R_1st DIE FPCB ALIGN BACKWARD
AND       F0009A
LOAD      T1069	// R_4th DIE ALIGN FORWARD
AND       P00063	// R_4th DIE FPCB ALIGN FORWARD
OR LOAD
AND LOAD
LOAD      F0009A
AND       T1800	// R-4th-Cyl-Align Out
OR        T1801	// R-4th-Cyl-Align In
AND LOAD
AND       T1802	// R-4th-Cyl-Side-Align Out
AND       P00140	// R_4th DIE VACUUM EJECTOR ON
OUT       M14034	// 09_Z move bending pos
// output comment: 09_ÀÚµ¿ ¾ó¶óÀÎ ÈÄÁø »çÀÌµå ¾ó¶óÀÎ ÈÄÁø
; L101
LOAD      M04203	// R_4th BD Z BENDING POS 2-ax20
LOAD      T1066	// R_1st DIE ALIGN BACKWARD
AND       T1068	// R_1st DIE FPCB ALIGN BACKWARD
AND       F0009A
LOAD      T1069	// R_4th DIE ALIGN FORWARD
AND       P00063	// R_4th DIE FPCB ALIGN FORWARD
OR LOAD
AND LOAD
LOAD      F0009A
AND       T1800	// R-4th-Cyl-Align Out
OR        T1801	// R-4th-Cyl-Align In
AND LOAD
AND       T1802	// R-4th-Cyl-Side-Align Out
AND       P00140	// R_4th DIE VACUUM EJECTOR ON
OUT       M14035	// 09_Z move bending pos 2
// output comment: 09_ÀÚµ¿ Z º¥µù À§Ä¡ ->
; L103
LOAD      M04203	// R_4th BD Z BENDING POS 2-ax20
LOAD      T1066	// R_1st DIE ALIGN BACKWARD
AND       T1068	// R_1st DIE FPCB ALIGN BACKWARD
AND       F0009A
LOAD      T1069	// R_4th DIE ALIGN FORWARD
AND       P00063	// R_4th DIE FPCB ALIGN FORWARD
OR LOAD
AND LOAD
AND       T1801	// R-4th-Cyl-Align In
AND       T1802	// R-4th-Cyl-Side-Align Out
AND       P00140	// R_4th DIE VACUUM EJECTOR ON
OUT       M14036	// 09_Cyl align In
// output comment: 09_ÀÚµ¿ »çÀÌµå ÆÝÄ¡ ÀüÁø
; L105
LOAD      M04203	// R_4th BD Z BENDING POS 2-ax20
LOAD      T1066	// R_1st DIE ALIGN BACKWARD
AND       T1068	// R_1st DIE FPCB ALIGN BACKWARD
AND       F0009A
LOAD      T1069	// R_4th DIE ALIGN FORWARD
AND       P00063	// R_4th DIE FPCB ALIGN FORWARD
OR LOAD
AND LOAD
AND       T1801	// R-4th-Cyl-Align In
AND       T1803	// R-4th-Cyl-Side-Align In
AND       P00140	// R_4th DIE VACUUM EJECTOR ON
OUT       M14037	// 09_Cyl side align in
// output comment: 09_ÀÚµ¿ »çÀÌµå ÆÝÄ¡ ÈÄÁø(X1652) 09_ÀÚµ¿ Z »ó½Â À§Ä¡ -> (X1666)

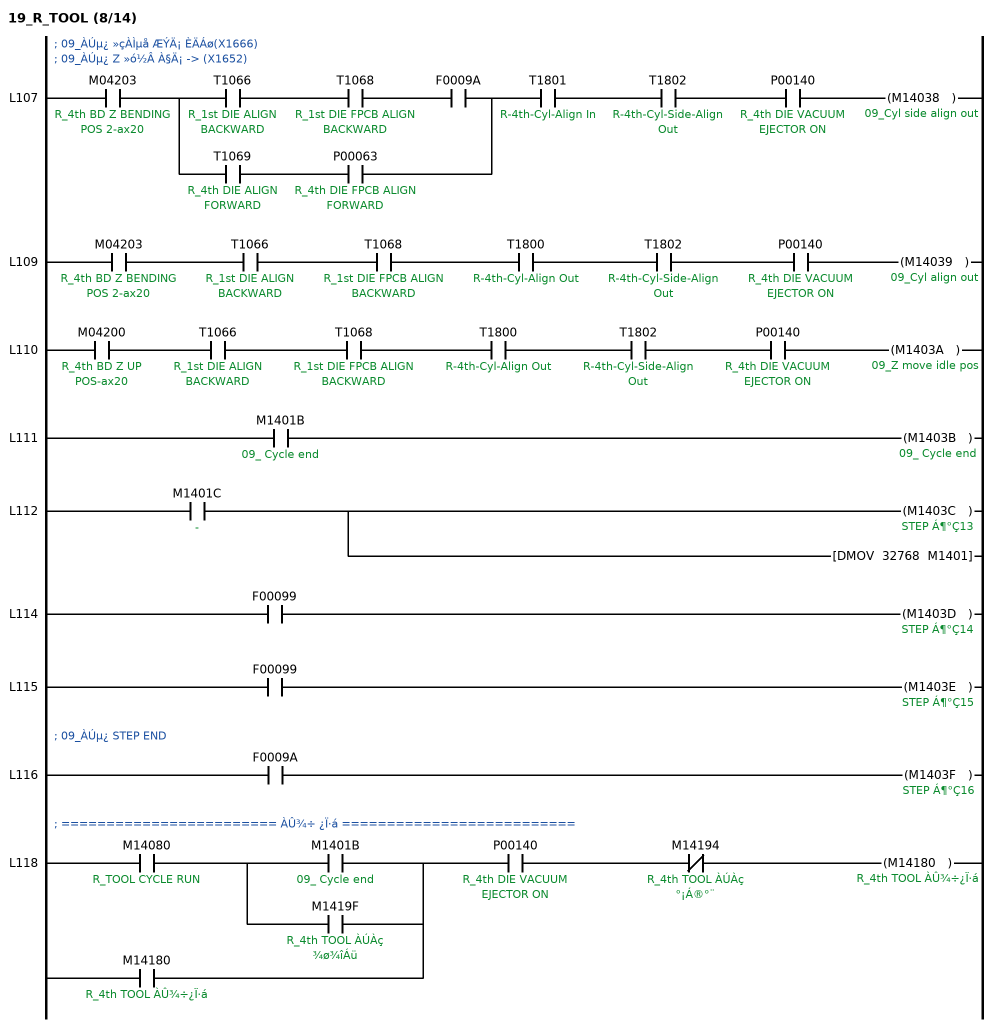
; L107
LOAD      M04203	// R_4th BD Z BENDING POS 2-ax20
LOAD      T1066	// R_1st DIE ALIGN BACKWARD
AND       T1068	// R_1st DIE FPCB ALIGN BACKWARD
AND       F0009A
LOAD      T1069	// R_4th DIE ALIGN FORWARD
AND       P00063	// R_4th DIE FPCB ALIGN FORWARD
OR LOAD
AND LOAD
AND       T1801	// R-4th-Cyl-Align In
AND       T1802	// R-4th-Cyl-Side-Align Out
AND       P00140	// R_4th DIE VACUUM EJECTOR ON
OUT       M14038	// 09_Cyl side align out
// output comment: 09_ÀÚµ¿ »çÀÌµå ÆÝÄ¡ ÈÄÁø(X1666) 09_ÀÚµ¿ Z »ó½Â À§Ä¡ -> (X1652)
; L109
LOAD      M04203	// R_4th BD Z BENDING POS 2-ax20
AND       T1066	// R_1st DIE ALIGN BACKWARD
AND       T1068	// R_1st DIE FPCB ALIGN BACKWARD
AND       T1800	// R-4th-Cyl-Align Out
AND       T1802	// R-4th-Cyl-Side-Align Out
AND       P00140	// R_4th DIE VACUUM EJECTOR ON
OUT       M14039	// 09_Cyl align out
; L110
LOAD      M04200	// R_4th BD Z UP POS-ax20
AND       T1066	// R_1st DIE ALIGN BACKWARD
AND       T1068	// R_1st DIE FPCB ALIGN BACKWARD
AND       T1800	// R-4th-Cyl-Align Out
AND       T1802	// R-4th-Cyl-Side-Align Out
AND       P00140	// R_4th DIE VACUUM EJECTOR ON
OUT       M1403A	// 09_Z move idle pos
; L111
LOAD      M1401B	// 09_ Cycle end
OUT       M1403B	// 09_ Cycle end
; L112
LOAD      M1401C	// -
OUT       M1403C	// STEP Á¶°Ç13
DMOV      32768 M1401
; L114
LOAD      F00099
OUT       M1403D	// STEP Á¶°Ç14
; L115
LOAD      F00099
OUT       M1403E	// STEP Á¶°Ç15
; L116
LOAD      F0009A
OUT       M1403F	// STEP Á¶°Ç16
// output comment: 09_ÀÚµ¿ STEP END
// ======================== ÀÛ¾÷ ¿Ï·á ==========================
; L118
LOAD      M14080	// R_TOOL CYCLE RUN
LOAD      M1401B	// 09_ Cycle end
OR        M1419F	// R_4th TOOL ÀÚÀç ¾ø¾îÁü
AND LOAD
OR        M14180	// R_4th TOOL ÀÛ¾÷¿Ï·á
AND       P00140	// R_4th DIE VACUUM EJECTOR ON
AND NOT   M14194	// R_4th TOOL ÀÚÀç °¡Á®°¨
OUT       M14180	// R_4th TOOL ÀÛ¾÷¿Ï·á

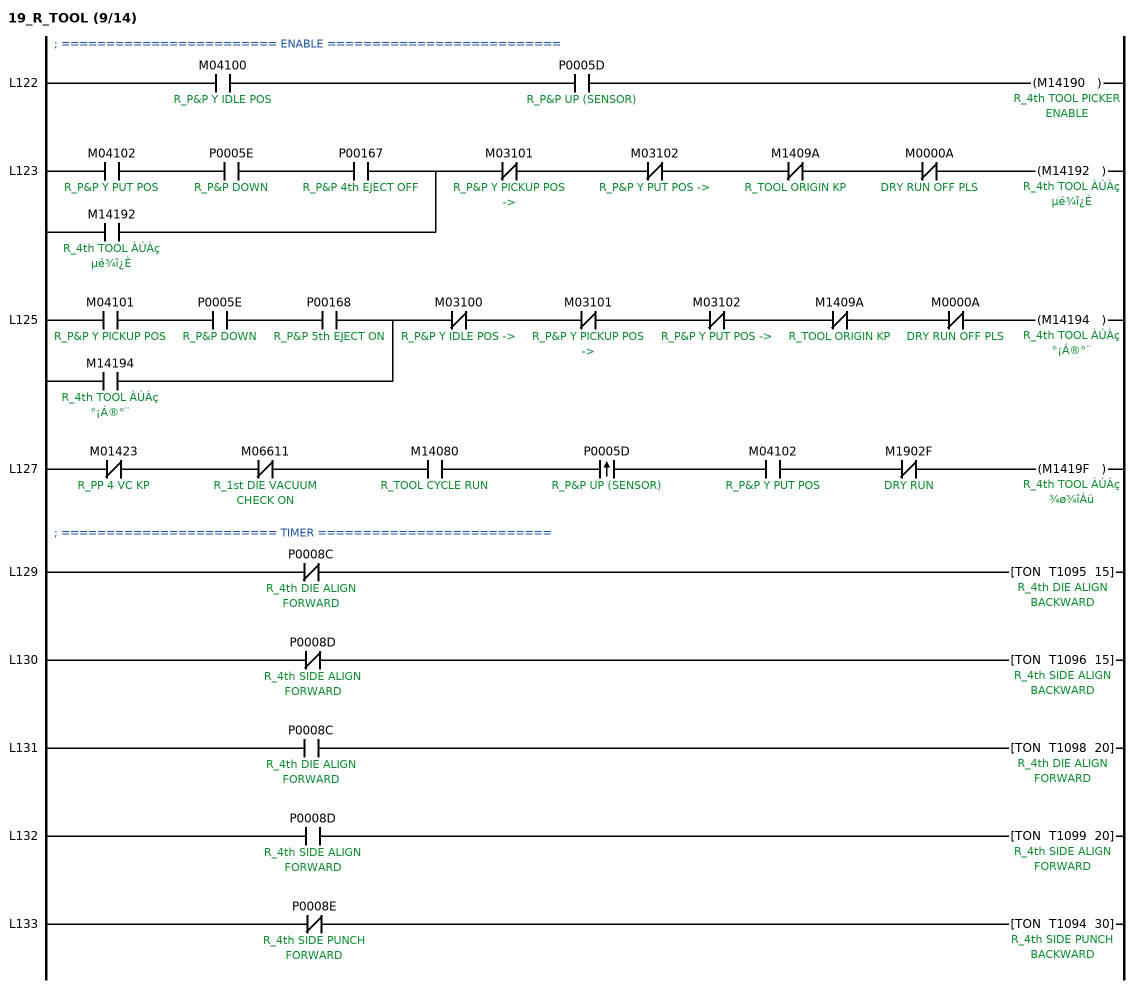
// ======================== ENABLE ==========================
; L122
LOAD      M04100	// R_P&P Y IDLE POS
AND       P0005D	// R_P&P UP (SENSOR)
OUT       M14190	// R_4th TOOL PICKER ENABLE
; L123
LOAD      M04102	// R_P&P Y PUT POS
AND       P0005E	// R_P&P DOWN
AND       P00167	// R_P&P 4th EJECT OFF
OR        M14192	// R_4th TOOL ÀÚÀç µé¾î¿È
AND NOT   M03101	// R_P&P Y PICKUP POS ->
AND NOT   M03102	// R_P&P Y PUT POS ->
AND NOT   M1409A	// R_TOOL ORIGIN KP
AND NOT   M0000A	// DRY RUN OFF PLS
OUT       M14192	// R_4th TOOL ÀÚÀç µé¾î¿È
; L125
LOAD      M04101	// R_P&P Y PICKUP POS
AND       P0005E	// R_P&P DOWN
AND       P00168	// R_P&P 5th EJECT ON
OR        M14194	// R_4th TOOL ÀÚÀç °¡Á®°¨
AND NOT   M03100	// R_P&P Y IDLE POS ->
AND NOT   M03101	// R_P&P Y PICKUP POS ->
AND NOT   M03102	// R_P&P Y PUT POS ->
AND NOT   M1409A	// R_TOOL ORIGIN KP
AND NOT   M0000A	// DRY RUN OFF PLS
OUT       M14194	// R_4th TOOL ÀÚÀç °¡Á®°¨
; L127
LOAD NOT  M01423	// R_PP 4 VC KP
AND NOT   M06611	// R_1st DIE VACUUM CHECK ON
AND       M14080	// R_TOOL CYCLE RUN
ANDP      P0005D	// R_P&P UP (SENSOR)
AND       M04102	// R_P&P Y PUT POS
AND NOT   M1902F	// DRY RUN
OUT       M1419F	// R_4th TOOL ÀÚÀç ¾ø¾îÁü
// ======================== TIMER ==========================
; L129
LOAD NOT  P0008C	// R_4th DIE ALIGN FORWARD
TON       T1095 15	// R_4th DIE ALIGN BACKWARD
; L130
LOAD NOT  P0008D	// R_4th SIDE ALIGN FORWARD
TON       T1096 15	// R_4th SIDE ALIGN BACKWARD
; L131
LOAD      P0008C	// R_4th DIE ALIGN FORWARD
TON       T1098 20	// R_4th DIE ALIGN FORWARD
; L132
LOAD      P0008D	// R_4th SIDE ALIGN FORWARD
TON       T1099 20	// R_4th SIDE ALIGN FORWARD
; L133
LOAD NOT  P0008E	// R_4th SIDE PUNCH FORWARD
TON       T1094 30	// R_4th SIDE PUNCH BACKWARD

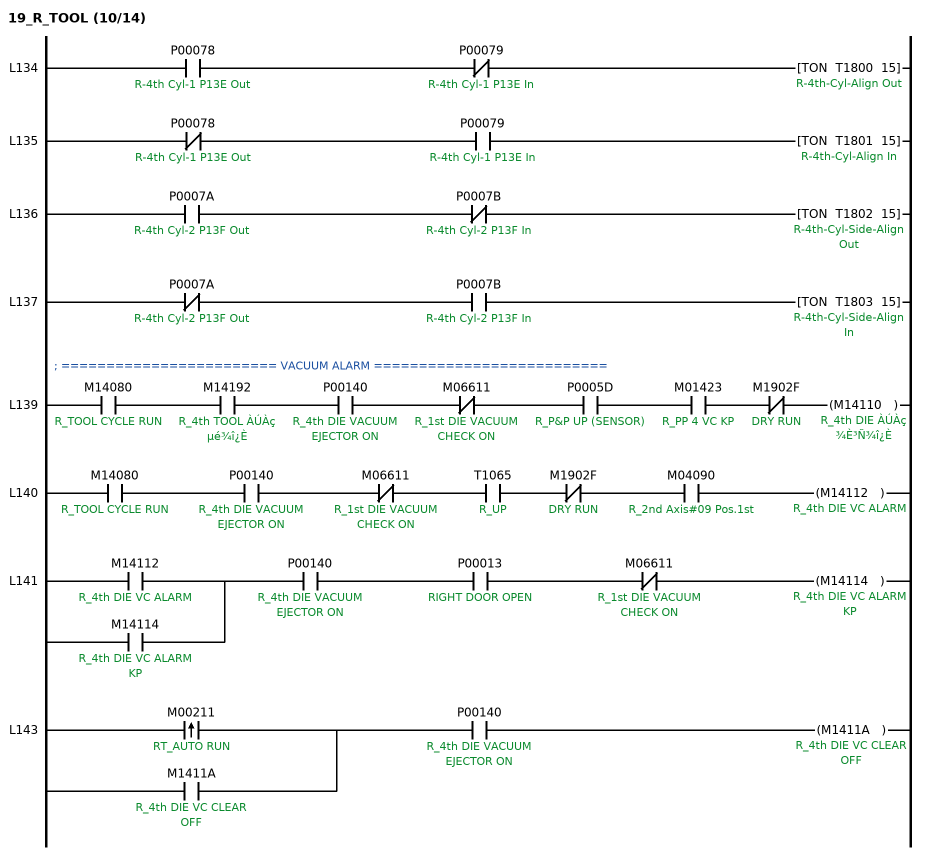
; L134
LOAD      P00078	// R-4th Cyl-1 P13E Out
AND NOT   P00079	// R-4th Cyl-1 P13E In
TON       T1800 15	// R-4th-Cyl-Align Out
; L135
LOAD NOT  P00078	// R-4th Cyl-1 P13E Out
AND       P00079	// R-4th Cyl-1 P13E In
TON       T1801 15	// R-4th-Cyl-Align In
; L136
LOAD      P0007A	// R-4th Cyl-2 P13F Out
AND NOT   P0007B	// R-4th Cyl-2 P13F In
TON       T1802 15	// R-4th-Cyl-Side-Align Out
; L137
LOAD NOT  P0007A	// R-4th Cyl-2 P13F Out
AND       P0007B	// R-4th Cyl-2 P13F In
TON       T1803 15	// R-4th-Cyl-Side-Align In
// ======================== VACUUM ALARM ==========================
; L139
LOAD      M14080	// R_TOOL CYCLE RUN
AND       M14192	// R_4th TOOL ÀÚÀç µé¾î¿È
AND       P00140	// R_4th DIE VACUUM EJECTOR ON
AND NOT   M06611	// R_1st DIE VACUUM CHECK ON
AND       P0005D	// R_P&P UP (SENSOR)
AND       M01423	// R_PP 4 VC KP
AND NOT   M1902F	// DRY RUN
OUT       M14110	// R_4th DIE ÀÚÀç ¾È³Ñ¾î¿È
; L140
LOAD      M14080	// R_TOOL CYCLE RUN
AND       P00140	// R_4th DIE VACUUM EJECTOR ON
AND NOT   M06611	// R_1st DIE VACUUM CHECK ON
AND       T1065	// R_UP
AND NOT   M1902F	// DRY RUN
AND       M04090	// R_2nd Axis#09 Pos.1st
OUT       M14112	// R_4th DIE VC ALARM
; L141
LOAD      M14112	// R_4th DIE VC ALARM
OR        M14114	// R_4th DIE VC ALARM KP
AND       P00140	// R_4th DIE VACUUM EJECTOR ON
AND       P00013	// RIGHT DOOR OPEN
AND NOT   M06611	// R_1st DIE VACUUM CHECK ON
OUT       M14114	// R_4th DIE VC ALARM KP
; L143
LOADP     M00211	// RT_AUTO RUN
OR        M1411A	// R_4th DIE VC CLEAR OFF
AND       P00140	// R_4th DIE VACUUM EJECTOR ON
OUT       M1411A	// R_4th DIE VC CLEAR OFF

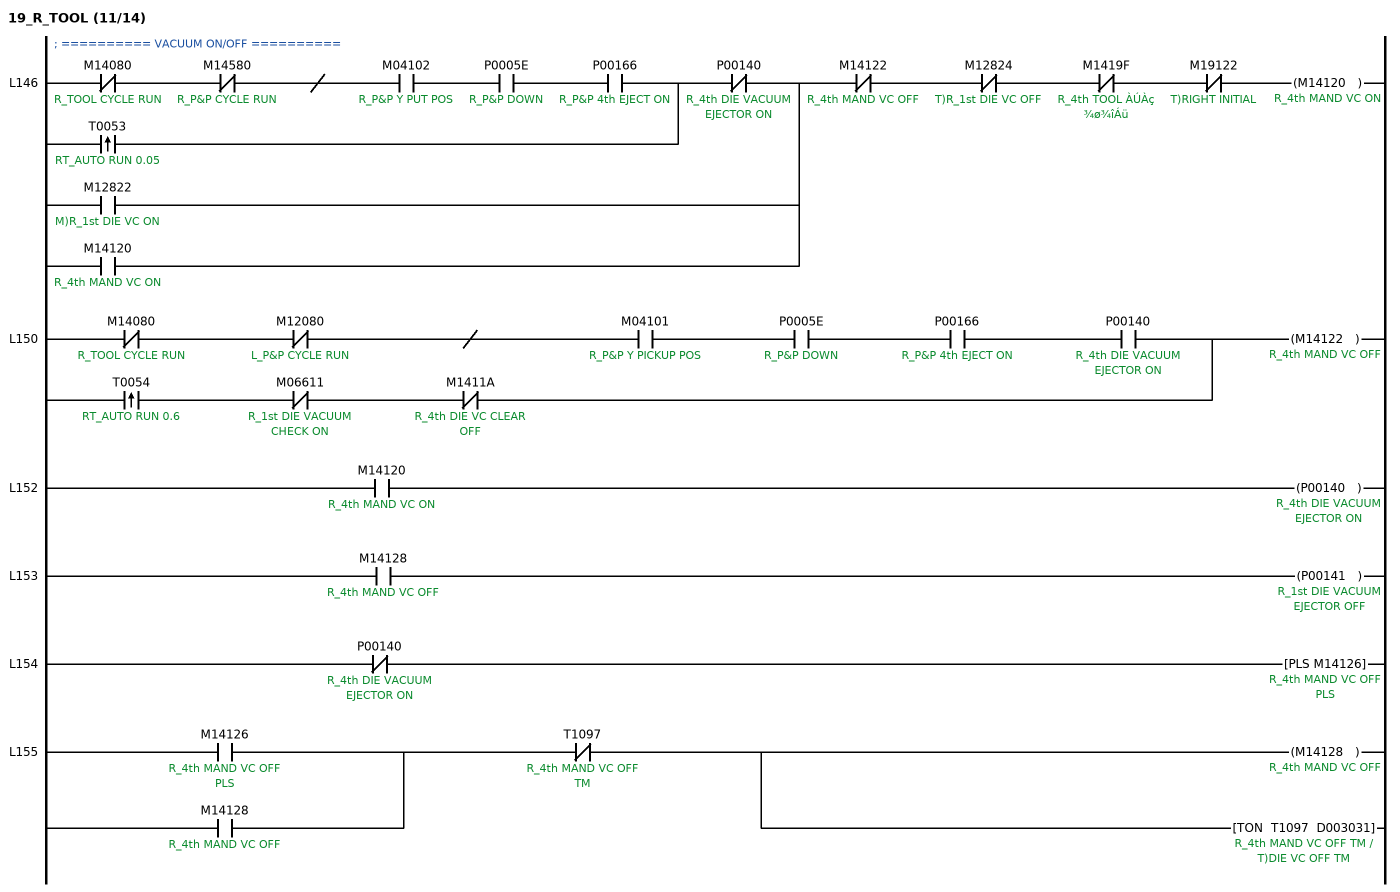
// ========== VACUUM ON/OFF ==========
; L146
LOAD NOT  M14080	// R_TOOL CYCLE RUN
AND NOT   M14580	// R_P&P CYCLE RUN
NOT
AND       M04102	// R_P&P Y PUT POS
AND       P0005E	// R_P&P DOWN
AND       P00166	// R_P&P 4th EJECT ON
ORP       T0053	// RT_AUTO RUN 0.05
AND NOT   P00140	// R_4th DIE VACUUM EJECTOR ON
OR        M12822	// M)R_1st DIE VC ON
OR        M14120	// R_4th MAND VC ON
AND NOT   M14122	// R_4th MAND VC OFF
AND NOT   M12824	// T)R_1st DIE VC OFF
AND NOT   M1419F	// R_4th TOOL ÀÚÀç ¾ø¾îÁü
AND NOT   M19122	// T)RIGHT INITIAL
OUT       M14120	// R_4th MAND VC ON
; L150
LOAD NOT  M14080	// R_TOOL CYCLE RUN
AND NOT   M12080	// L_P&P CYCLE RUN
NOT
AND       M04101	// R_P&P Y PICKUP POS
AND       P0005E	// R_P&P DOWN
AND       P00166	// R_P&P 4th EJECT ON
AND       P00140	// R_4th DIE VACUUM EJECTOR ON
LOADP     T0054	// RT_AUTO RUN 0.6
AND NOT   M06611	// R_1st DIE VACUUM CHECK ON
AND NOT   M1411A	// R_4th DIE VC CLEAR OFF
OR LOAD
OUT       M14122	// R_4th MAND VC OFF
; L152
LOAD      M14120	// R_4th MAND VC ON
OUT       P00140	// R_4th DIE VACUUM EJECTOR ON
; L153
LOAD      M14128	// R_4th MAND VC OFF
OUT       P00141	// R_1st DIE VACUUM EJECTOR OFF
; L154
LOAD NOT  P00140	// R_4th DIE VACUUM EJECTOR ON
OUTP      M14126	// R_4th MAND VC OFF PLS
; L155
LOAD      M14126	// R_4th MAND VC OFF PLS
OR        M14128	// R_4th MAND VC OFF
AND NOT   T1097	// R_4th MAND VC OFF TM
OUT       M14128	// R_4th MAND VC OFF
TON       T1097 D003031	// R_4th MAND VC OFF TM / T)DIE VC OFF TM

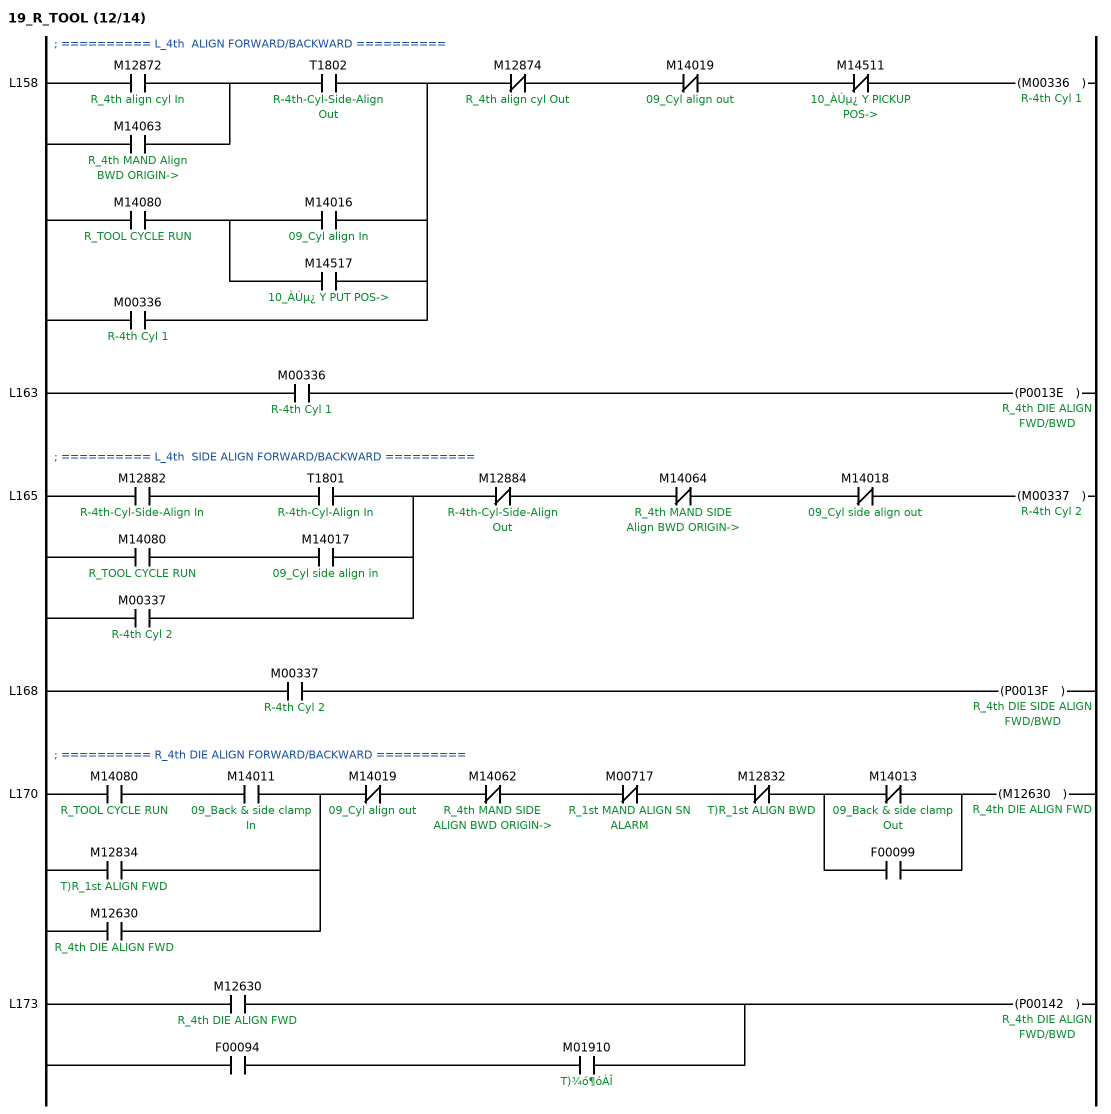
// ========== L_4th  ALIGN FORWARD/BACKWARD ==========
; L158
LOAD      M12872	// R_4th align cyl In
OR        M14063	// R_4th MAND Align BWD ORIGIN->
AND       T1802	// R-4th-Cyl-Side-Align Out
LOAD      M14080	// R_TOOL CYCLE RUN
LOAD      M14016	// 09_Cyl align In
OR        M14517	// 10_ÀÚµ¿ Y PUT POS->
AND LOAD
OR LOAD
OR        M00336	// R-4th Cyl 1
AND NOT   M12874	// R_4th align cyl Out
AND NOT   M14019	// 09_Cyl align out
AND NOT   M14511	// 10_ÀÚµ¿ Y PICKUP POS->
OUT       M00336	// R-4th Cyl 1
; L163
LOAD      M00336	// R-4th Cyl 1
OUT       P0013E	// R_4th DIE ALIGN FWD/BWD
// ========== L_4th  SIDE ALIGN FORWARD/BACKWARD ==========
; L165
LOAD      M12882	// R-4th-Cyl-Side-Align In
AND       T1801	// R-4th-Cyl-Align In
LOAD      M14080	// R_TOOL CYCLE RUN
AND       M14017	// 09_Cyl side align in
OR LOAD
OR        M00337	// R-4th Cyl 2
AND NOT   M12884	// R-4th-Cyl-Side-Align Out
AND NOT   M14064	// R_4th MAND SIDE Align BWD ORIGIN->
AND NOT   M14018	// 09_Cyl side align out
OUT       M00337	// R-4th Cyl 2
; L168
LOAD      M00337	// R-4th Cyl 2
OUT       P0013F	// R_4th DIE SIDE ALIGN FWD/BWD
// ========== R_4th DIE ALIGN FORWARD/BACKWARD ==========
; L170
LOAD      M14080	// R_TOOL CYCLE RUN
AND       M14011	// 09_Back & side clamp In
OR        M12834	// T)R_1st ALIGN FWD
OR        M12630	// R_4th DIE ALIGN FWD
AND NOT   M14019	// 09_Cyl align out
AND NOT   M14062	// R_4th MAND SIDE ALIGN BWD ORIGIN->
AND NOT   M00717	// R_1st MAND ALIGN SN ALARM
AND NOT   M12832	// T)R_1st ALIGN BWD
LOAD NOT  M14013	// 09_Back & side clamp Out
OR        F00099
AND LOAD
OUT       M12630	// R_4th DIE ALIGN FWD
; L173
LOAD      M12630	// R_4th DIE ALIGN FWD
LOAD      F00094
AND       M01910	// T)¾ó¶óÀÎ
OR LOAD
OUT       P00142	// R_4th DIE ALIGN FWD/BWD

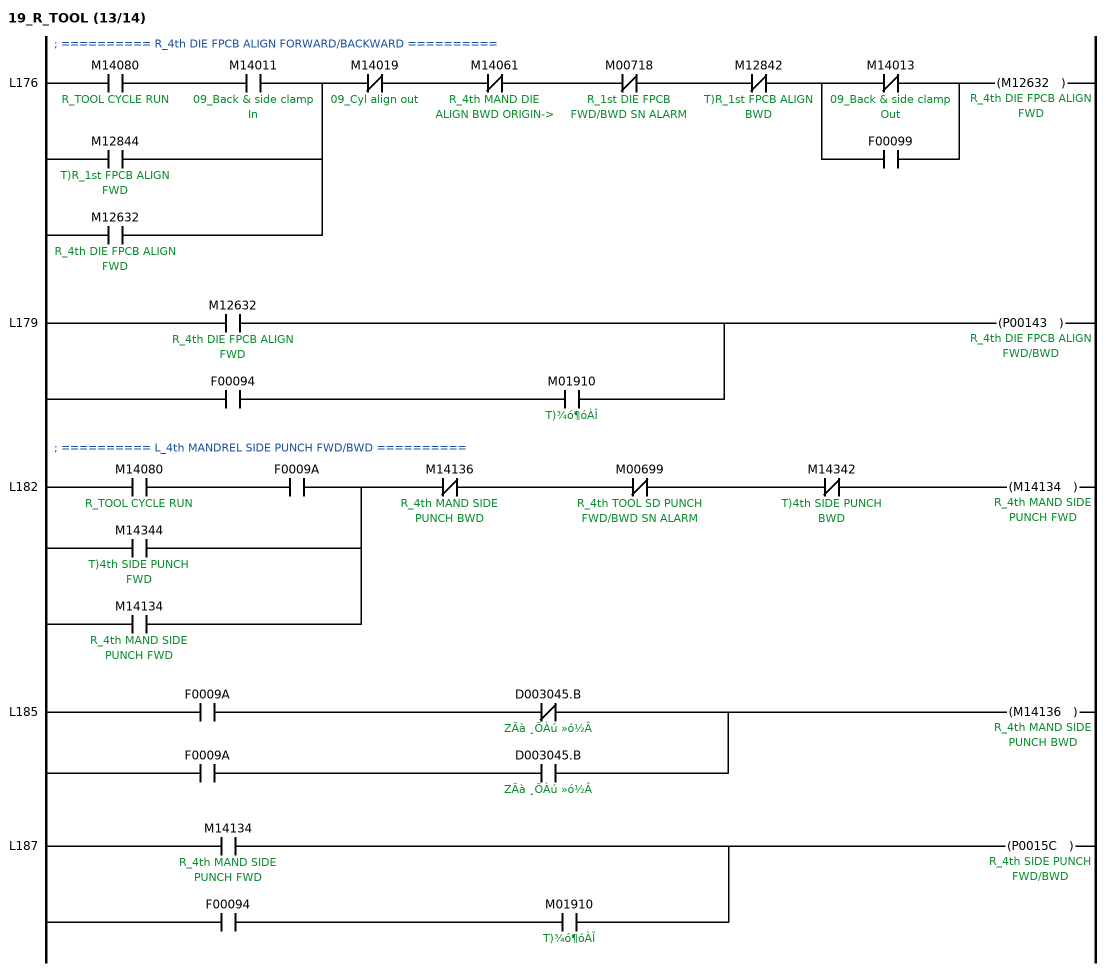
// ========== R_4th DIE FPCB ALIGN FORWARD/BACKWARD ==========
; L176
LOAD      M14080	// R_TOOL CYCLE RUN
AND       M14011	// 09_Back & side clamp In
OR        M12844	// T)R_1st FPCB ALIGN FWD
OR        M12632	// R_4th DIE FPCB ALIGN FWD
AND NOT   M14019	// 09_Cyl align out
AND NOT   M14061	// R_4th MAND DIE ALIGN BWD ORIGIN->
AND NOT   M00718	// R_1st DIE FPCB FWD/BWD SN ALARM
AND NOT   M12842	// T)R_1st FPCB ALIGN BWD
LOAD NOT  M14013	// 09_Back & side clamp Out
OR        F00099
AND LOAD
OUT       M12632	// R_4th DIE FPCB ALIGN FWD
; L179
LOAD      M12632	// R_4th DIE FPCB ALIGN FWD
LOAD      F00094
AND       M01910	// T)¾ó¶óÀÎ
OR LOAD
OUT       P00143	// R_4th DIE FPCB ALIGN FWD/BWD
// ========== L_4th MANDREL SIDE PUNCH FWD/BWD ==========
; L182
LOAD      M14080	// R_TOOL CYCLE RUN
AND       F0009A
OR        M14344	// T)4th SIDE PUNCH FWD
OR        M14134	// R_4th MAND SIDE PUNCH FWD
AND NOT   M14136	// R_4th MAND SIDE PUNCH BWD
AND NOT   M00699	// R_4th TOOL SD PUNCH FWD/BWD SN ALARM
AND NOT   M14342	// T)4th SIDE PUNCH BWD
OUT       M14134	// R_4th MAND SIDE PUNCH FWD
; L185
LOAD      F0009A
AND NOT   D003045.B	// ZÃà ¸ÕÀú »ó½Â
LOAD      F0009A
AND       D003045.B	// ZÃà ¸ÕÀú »ó½Â
OR LOAD
OUT       M14136	// R_4th MAND SIDE PUNCH BWD
; L187
LOAD      M14134	// R_4th MAND SIDE PUNCH FWD
LOAD      F00094
AND       M01910	// T)¾ó¶óÀÎ
OR LOAD
OUT       P0015C	// R_4th SIDE PUNCH FWD/BWD

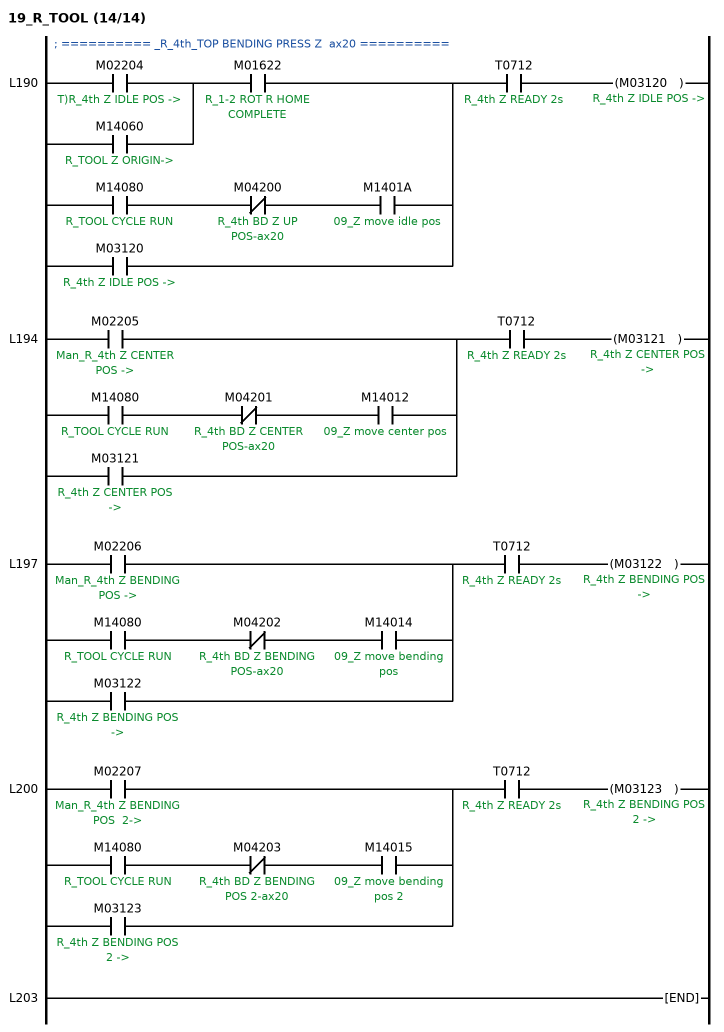
// ========== _R_4th_TOP BENDING PRESS Z  ax20 ==========
; L190
LOAD      M02204	// T)R_4th Z IDLE POS ->
OR        M14060	// R_TOOL Z ORIGIN->
AND       M01622	// R_1-2 ROT R HOME COMPLETE
LOAD      M14080	// R_TOOL CYCLE RUN
AND NOT   M04200	// R_4th BD Z UP POS-ax20
AND       M1401A	// 09_Z move idle pos
OR LOAD
OR        M03120	// R_4th Z IDLE POS ->
AND       T0712	// R_4th Z READY 2s
OUT       M03120	// R_4th Z IDLE POS ->
; L194
LOAD      M02205	// Man_R_4th Z CENTER POS ->
LOAD      M14080	// R_TOOL CYCLE RUN
AND NOT   M04201	// R_4th BD Z CENTER POS-ax20
AND       M14012	// 09_Z move center pos
OR LOAD
OR        M03121	// R_4th Z CENTER POS ->
AND       T0712	// R_4th Z READY 2s
OUT       M03121	// R_4th Z CENTER POS ->
; L197
LOAD      M02206	// Man_R_4th Z BENDING POS ->
LOAD      M14080	// R_TOOL CYCLE RUN
AND NOT   M04202	// R_4th BD Z BENDING POS-ax20
AND       M14014	// 09_Z move bending pos
OR LOAD
OR        M03122	// R_4th Z BENDING POS ->
AND       T0712	// R_4th Z READY 2s
OUT       M03122	// R_4th Z BENDING POS ->
; L200
LOAD      M02207	// Man_R_4th Z BENDING POS  2->
LOAD      M14080	// R_TOOL CYCLE RUN
AND NOT   M04203	// R_4th BD Z BENDING POS 2-ax20
AND       M14015	// 09_Z move bending pos 2
OR LOAD
OR        M03123	// R_4th Z BENDING POS 2 ->
AND       T0712	// R_4th Z READY 2s
OUT       M03123	// R_4th Z BENDING POS 2 ->
; L203
END

PROGRAM 20_R_PP (task: ½ºÄµ ÇÁ·Î±×·¥)

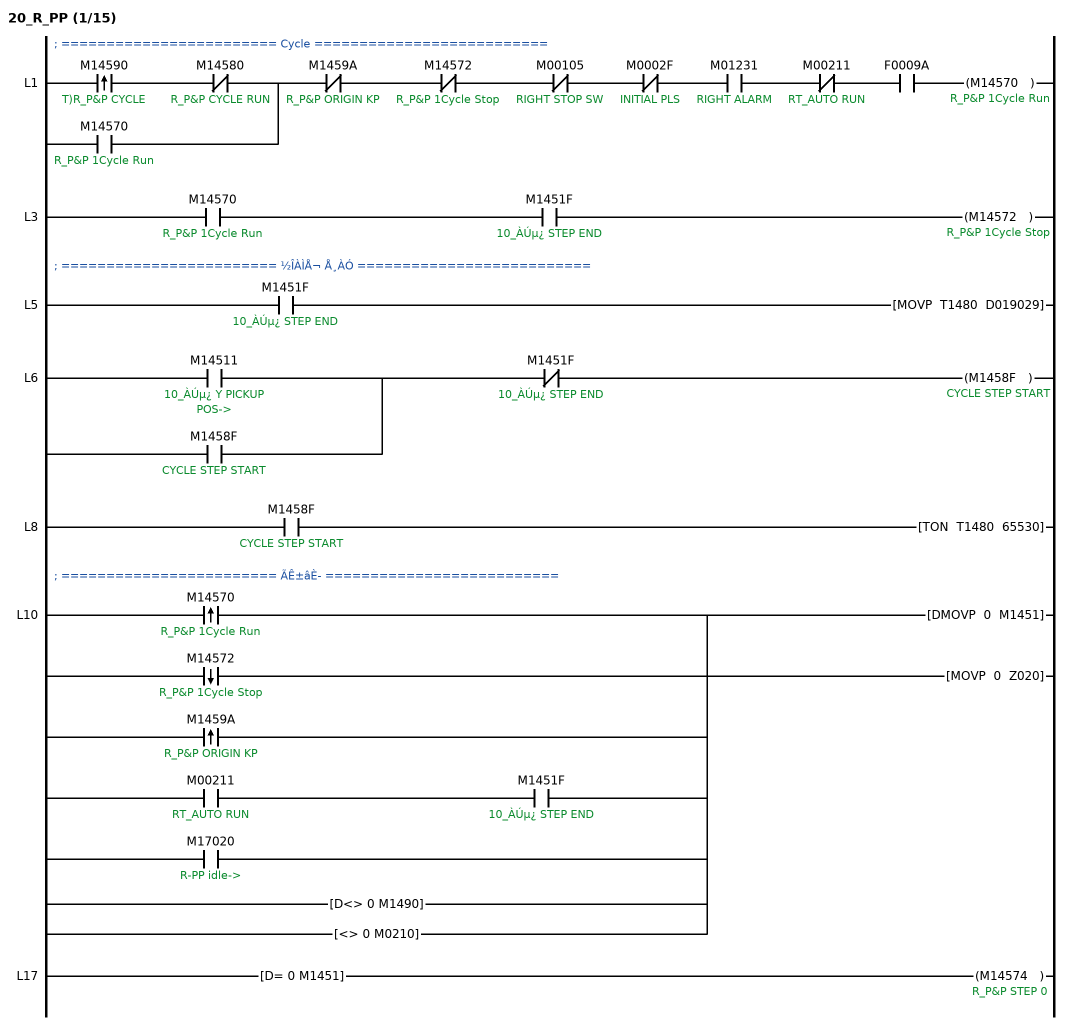
// ======================== Cycle ==========================
; L1
LOADP     M14590	// T)R_P&P CYCLE
AND NOT   M14580	// R_P&P CYCLE RUN
OR        M14570	// R_P&P 1Cycle Run
AND NOT   M1459A	// R_P&P ORIGIN KP
AND NOT   M14572	// R_P&P 1Cycle Stop
AND NOT   M00105	// RIGHT STOP SW
AND NOT   M0002F	// INITIAL PLS
AND       M01231	// RIGHT ALARM
AND NOT   M00211	// RT_AUTO RUN
AND       F0009A
OUT       M14570	// R_P&P 1Cycle Run
; L3
LOAD      M14570	// R_P&P 1Cycle Run
AND       M1451F	// 10_ÀÚµ¿ STEP END
OUT       M14572	// R_P&P 1Cycle Stop
// ======================== ½ÎÀÌÅ¬ Å¸ÀÓ ==========================
; L5
LOAD      M1451F	// 10_ÀÚµ¿ STEP END
MOVP      T1480 D019029
; L6
LOAD      M14511	// 10_ÀÚµ¿ Y PICKUP POS->
OR        M1458F	// CYCLE STEP START
AND NOT   M1451F	// 10_ÀÚµ¿ STEP END
OUT       M1458F	// CYCLE STEP START
; L8
LOAD      M1458F	// CYCLE STEP START
TON       T1480 65530
// ======================== ÃÊ±âÈ­ ==========================
; L10
LOADP     M14570	// R_P&P 1Cycle Run
ORN       M14572	// R_P&P 1Cycle Stop
ORP       M1459A	// R_P&P ORIGIN KP
LOAD      M00211	// RT_AUTO RUN
AND       M1451F	// 10_ÀÚµ¿ STEP END
OR LOAD
OR        M17020	// R-PP idle->
ORD<>     0 M1490
OR<>      0 M0210
DMOVP     0 M1451
MOVP      0 Z020
; L17
LOADD=    0 M1451
OUT       M14574	// R_P&P STEP 0

